C01828=1213.593,-33.093,-40.651,-179.967,5.450,148.943
C01829=1213.588,-32.844,-40.663,-179.964,5.451,148.942
C01830=1213.583,-32.594,-40.675,-179.962,5.450,148.942
C01831=1213.578,-32.344,-40.688,-179.960,5.451,148.941
C01832=1213.572,-32.095,-40.701,-179.957,5.451,148.940
C01833=1213.567,-31.845,-40.714,-179.955,5.451,148.940
C01834=1213.563,-31.595,-40.727,-179.953,5.452,148.939
C01835=1213.558,-31.347,-40.740,-179.950,5.452,148.939
C01836=1213.552,-31.097,-40.753,-179.948,5.452,148.938
C01837=1213.548,-30.847,-40.766,-179.945,5.452,148.937
C01838=1213.542,-30.598,-40.779,-179.943,5.453,148.936
C01839=1213.537,-30.348,-40.791,-179.941,5.453,148.936
C01840=1213.532,-30.098,-40.805,-179.938,5.453,148.935
C01841=1213.527,-29.849,-40.818,-179.935,5.454,148.934
C01842=1213.522,-29.599,-40.830,-179.933,5.454,148.934
C01843=1213.517,-29.349,-40.844,-179.931,5.454,148.933
C01844=1213.511,-29.100,-40.856,-179.928,5.454,148.932
C01845=1213.506,-28.850,-40.869,-179.925,5.455,148.932
C01846=1213.501,-28.600,-40.883,-179.923,5.454,148.931
C01847=1213.496,-28.351,-40.895,-179.921,5.455,148.930
C01848=1213.491,-28.101,-40.908,-179.918,5.456,148.930
C01849=1213.486,-27.852,-40.922,-179.916,5.455,148.929
C01850=1213.481,-27.602,-40.935,-179.914,5.456,148.928
C01851=1213.476,-27.352,-40.948,-179.911,5.456,148.928
C01852=1213.470,-27.103,-40.961,-179.908,5.457,148.927
C01853=1213.465,-26.853,-40.973,-179.906,5.456,148.926
C01854=1213.461,-26.603,-40.986,-179.904,5.457,148.925
C01855=1213.455,-26.354,-41.000,-179.901,5.457,148.925
C01856=1213.451,-26.104,-41.013,-179.899,5.457,148.924
C01857=1213.446,-25.855,-41.026,-179.896,5.458,148.923
C01858=1213.440,-25.605,-41.039,-179.893,5.458,148.923
C01859=1213.435,-25.355,-41.052,-179.891,5.458,148.922
C01860=1213.429,-25.106,-41.065,-179.889,5.458,148.921
C01861=1213.425,-24.856,-41.079,-179.887,5.459,148.921
C01862=1213.420,-24.607,-41.091,-179.884,5.460,148.920
C01863=1213.414,-24.357,-41.105,-179.882,5.459,148.919
C01864=1213.410,-24.107,-41.118,-179.879,5.460,148.919
C01865=1213.404,-23.858,-41.132,-179.877,5.460,148.918
C01866=1213.399,-23.608,-41.145,-179.874,5.460,148.917
C01867=1213.394,-23.359,-41.157,-179.872,5.460,148.917
C01868=1213.389,-23.090,-41.172,-179.869,5.461,148.916
C01869=1213.383,-22.820,-41.186,-179.866,5.461,148.915
C01870=1213.378,-22.551,-41.200,-179.863,5.462,148.914
C01871=1213.372,-22.281,-41.215,-179.861,5.462,148.914
C01872=1213.368,-22.031,-41.228,-179.859,5.462,148.913
C01873=1213.362,-21.782,-41.242,-179.856,5.462,148.912
C01874=1213.357,-21.533,-41.254,-179.854,5.463,148.912
C01875=1213.352,-21.282,-41.268,-179.852,5.463,148.911
C01876=1213.347,-21.034,-41.281,-179.849,5.463,148.910
C01877=1213.342,-20.783,-41.295,-179.846,5.464,148.910
C01878=1213.336,-20.534,-41.307,-179.844,5.464,148.909
C01879=1213.332,-20.284,-41.321,-179.842,5.464,148.908
C01880=1213.326,-20.035,-41.334,-179.839,5.464,148.908
C01881=1213.321,-19.785,-41.348,-179.836,5.465,148.907
C01882=1213.316,-19.536,-41.361,-179.834,5.465,148.906
C01883=1213.311,-19.286,-41.375,-179.832,5.465,148.906
C01884=1213.306,-19.037,-41.388,-179.829,5.466,148.905
C01885=1213.301,-18.787,-41.401,-179.826,5.466,148.904
C01886=1213.295,-18.537,-41.415,-179.824,5.466,148.903
C01887=1213.291,-18.288,-41.428,-179.822,5.466,148.903
C01888=1213.285,-18.038,-41.441,-179.819,5.467,148.902
C01889=1213.281,-17.789,-41.455,-179.817,5.468,148.902
C01890=1213.275,-17.539,-41.468,-179.815,5.467,148.901
C01891=1213.270,-17.289,-41.481,-179.812,5.468,148.900
C01892=1213.265,-17.040,-41.495,-179.809,5.468,148.900
C01893=1213.260,-16.790,-41.508,-179.807,5.469,148.899
C01894=1213.255,-16.541,-41.522,-179.805,5.468,148.898
C01895=1213.250,-16.291,-41.536,-179.802,5.469,148.897
C01896=1213.245,-16.041,-41.549,-179.799,5.469,148.897
C01897=1213.239,-15.792,-41.563,-179.797,5.470,148.896
C01898=1213.235,-15.542,-41.576,-179.794,5.470,148.895
C01899=1213.229,-15.293,-41.589,-179.792,5.470,148.895
C01900=1213.224,-15.043,-41.604,-179.789,5.471,148.894
C01901=1213.219,-14.794,-41.616,-179.787,5.471,148.893
C01902=1213.214,-14.544,-41.631,-179.785,5.471,148.893
C01903=1213.208,-14.294,-41.644,-179.782,5.472,148.892
C01904=1213.204,-14.045,-41.657,-179.780,5.472,148.891
C01905=1213.199,-13.795,-41.672,-179.777,5.473,148.891
C01906=1213.194,-13.546,-41.684,-179.775,5.472,148.890
C01907=1213.189,-13.296,-41.699,-179.772,5.473,148.889
C01908=1213.183,-13.046,-41.712,-179.770,5.473,148.889
C01909=1213.179,-12.797,-41.725,-179.767,5.474,148.888
C01910=1213.174,-12.547,-41.739,-179.765,5.473,148.887
C01911=1213.168,-12.298,-41.753,-179.762,5.474,148.887
C01912=1213.164,-12.048,-41.767,-179.760,5.474,148.886
C01913=1213.158,-11.799,-41.780,-179.757,5.475,148.885
C01914=1213.153,-11.549,-41.794,-179.755,5.475,148.885
C01915=1213.149,-11.300,-41.808,-179.753,5.475,148.884
C01916=1213.143,-11.050,-41.821,-179.750,5.476,148.883
C01917=1213.138,-10.800,-41.835,-179.747,5.476,148.883
C01918=1213.132,-10.551,-41.848,-179.745,5.477,148.882
C01919=1213.128,-10.301,-41.862,-179.743,5.477,148.881
C01920=1213.123,-10.051,-41.876,-179.740,5.477,148.881
C01921=1213.117,-9.802,-41.890,-179.737,5.478,148.880
C01922=1213.113,-9.552,-41.903,-179.735,5.478,148.879
C01923=1213.108,-9.303,-41.918,-179.733,5.478,148.878
C01924=1213.103,-9.054,-41.931,-179.730,5.478,148.878
C01925=1213.097,-8.803,-41.945,-179.727,5.479,148.877
C01926=1213.093,-8.554,-41.959,-179.725,5.479,148.876
C01927=1213.088,-8.305,-41.973,-179.723,5.479,148.876
C01928=1213.082,-8.055,-41.986,-179.720,5.480,148.875
C01929=1213.077,-7.805,-42.000,-179.718,5.480,148.875
C01930=1213.072,-7.556,-42.014,-179.715,5.481,148.874
C01931=1213.068,-7.307,-42.028,-179.712,5.481,148.873
C01932=1213.062,-7.056,-42.042,-179.710,5.481,148.872
C01933=1213.057,-6.807,-42.056,-179.708,5.482,148.872
C01934=1213.052,-6.557,-42.070,-179.705,5.482,148.871
C01935=1213.048,-6.308,-42.084,-179.702,5.483,148.870
C01936=1213.042,-6.059,-42.097,-179.700,5.482,148.870
C01937=1213.037,-5.809,-42.111,-179.698,5.483,148.869
C01938=1213.032,-5.559,-42.125,-179.695,5.483,148.868
C01939=1213.027,-5.309,-42.140,-179.693,5.484,148.868
C01940=1213.021,-5.060,-42.153,-179.690,5.485,148.867
C01941=1213.017,-4.811,-42.167,-179.688,5.484,148.867
C01942=1213.012,-4.561,-42.181,-179.685,5.485,148.866
C01943=1213.006,-4.312,-42.195,-179.683,5.485,148.865
C01944=1213.001,-4.062,-42.209,-179.680,5.486,148.864
C01945=1212.996,-3.812,-42.223,-179.677,5.486,148.864
C01946=1212.991,-3.562,-42.237,-179.675,5.486,148.863
C01947=1212.986,-3.313,-42.251,-179.673,5.487,148.862
C01948=1212.982,-3.064,-42.265,-179.670,5.487,148.862
C01949=1212.977,-2.814,-42.279,-179.667,5.488,148.861
C01950=1212.971,-2.565,-42.293,-179.665,5.488,148.861
C01951=1212.966,-2.315,-42.307,-179.663,5.488,148.860
C01952=1212.961,-2.065,-42.321,-179.660,5.489,148.859
C01953=1212.956,-1.816,-42.335,-179.658,5.489,148.858
C01954=1212.950,-1.567,-42.349,-179.655,5.490,148.858
C01955=1212.945,-1.317,-42.364,-179.653,5.490,148.857
C01956=1212.941,-1.067,-42.378,-179.650,5.490,148.856
C01957=1212.936,-0.817,-42.392,-179.648,5.490,148.856
C01958=1212.931,-0.568,-42.406,-179.645,5.491,148.855
C01959=1212.926,-0.319,-42.420,-179.642,5.491,148.854
C01960=1212.921,-0.069,-42.434,-179.640,5.492,148.854
C01961=1212.916,0.180,-42.448,-179.638,5.492,148.853
C01962=1212.911,0.430,-42.462,-179.636,5.492,148.852
C01963=1212.905,0.679,-42.476,-179.633,5.493,148.852
C01964=1212.900,0.929,-42.491,-179.630,5.493,148.851
C01965=1212.895,1.179,-42.505,-179.628,5.494,148.850
C01966=1212.891,1.428,-42.519,-179.626,5.494,148.850
C01967=1212.886,1.678,-42.534,-179.623,5.494,148.849
C01968=1212.880,1.927,-42.547,-179.620,5.495,148.848
C01969=1212.875,2.177,-42.562,-179.618,5.495,148.848
C01970=1212.870,2.426,-42.576,-179.615,5.496,148.847
C01971=1212.865,2.676,-42.590,-179.612,5.496,148.846
C01972=1212.860,2.945,-42.606,-179.610,5.496,148.846
C01973=1212.855,3.214,-42.621,-179.608,5.496,148.845
C01974=1212.848,3.483,-42.637,-179.605,5.497,148.844
C01975=1212.843,3.751,-42.653,-179.602,5.497,148.844
C01976=1212.838,4.001,-42.667,-179.600,5.498,148.843
C01977=1212.833,4.251,-42.681,-179.597,5.498,148.842
C01978=1212.828,4.501,-42.695,-179.594,5.499,148.841
C01979=1212.823,4.750,-42.710,-179.592,5.499,148.841
C01980=1212.818,5.000,-42.724,-179.590,5.499,148.840
C01981=1212.813,5.249,-42.738,-179.587,5.500,148.840
C01982=1212.808,5.499,-42.752,-179.585,5.501,148.839
C01983=1212.803,5.748,-42.767,-179.582,5.501,148.838
C01984=1212.798,5.998,-42.781,-179.579,5.502,148.838
C01985=1212.793,6.247,-42.796,-179.577,5.502,148.837
C01986=1212.788,6.497,-42.810,-179.575,5.502,148.836
C01987=1212.783,6.747,-42.824,-179.572,5.502,148.836
C01988=1212.777,6.995,-42.840,-179.569,5.503,148.835
C01989=1212.772,7.245,-42.854,-179.567,5.503,148.834
C01990=1212.767,7.495,-42.868,-179.564,5.504,148.833
C01991=1212.762,7.745,-42.882,-179.562,5.505,148.833
C01992=1212.758,7.994,-42.897,-179.559,5.505,148.832
C01993=1212.753,8.243,-42.912,-179.557,5.505,148.832
C01994=1212.748,8.493,-42.926,-179.555,5.505,148.831
C01995=1212.743,8.743,-42.940,-179.552,5.506,148.830
C01996=1212.737,8.992,-42.956,-179.549,5.507,148.830
C01997=1212.733,9.242,-42.970,-179.547,5.507,148.829
C01998=1212.728,9.492,-42.984,-179.544,5.508,148.828
C01999=1212.722,9.741,-42.998,-179.542,5.507,148.828
C02000=1212.717,9.990,-43.013,-179.540,5.508,148.827
C02001=1212.712,10.239,-43.027,-179.537,5.509,148.826
C02002=1212.707,10.489,-43.042,-179.534,5.509,148.826
C02003=1212.702,10.739,-43.057,-179.532,5.510,148.825
C02004=1212.697,10.988,-43.072,-179.529,5.510,148.824
C02005=1212.692,11.238,-43.086,-179.527,5.511,148.824
C02006=1212.688,11.487,-43.101,-179.524,5.510,148.823
C02007=1212.682,11.737,-43.116,-179.522,5.511,148.822
C02008=1212.677,11.987,-43.130,-179.519,5.511,148.822
C02009=1212.672,12.236,-43.145,-179.517,5.512,148.821
C02010=1212.667,12.486,-43.159,-179.514,5.513,148.820
C02011=1212.663,12.735,-43.174,-179.512,5.513,148.820
C02012=1212.657,12.985,-43.189,-179.509,5.514,148.819
C02013=1212.652,13.234,-43.203,-179.507,5.514,148.818
C02014=1212.647,13.483,-43.218,-179.504,5.514,148.818
C02015=1212.642,13.733,-43.233,-179.502,5.515,148.817
C02016=1212.637,13.983,-43.248,-179.499,5.515,148.816
C02017=1212.632,14.232,-43.263,-179.496,5.516,148.816
C02018=1212.627,14.481,-43.278,-179.494,5.517,148.815
C02019=1212.622,14.731,-43.292,-179.492,5.517,148.815
C02020=1212.617,14.981,-43.307,-179.490,5.517,148.814
C02021=1212.612,15.230,-43.322,-179.487,5.517,148.813
C02022=1212.607,15.480,-43.336,-179.484,5.518,148.812
C02023=1212.602,15.729,-43.352,-179.482,5.518,148.812
C02024=1212.597,15.979,-43.366,-179.479,5.519,148.811
C02025=1212.592,16.228,-43.381,-179.476,5.519,148.810
C02026=1212.586,16.478,-43.396,-179.474,5.520,148.810
C02027=1212.582,16.727,-43.411,-179.471,5.521,148.809
C02028=1212.577,16.977,-43.425,-179.469,5.520,148.809
C02029=1212.571,17.226,-43.441,-179.467,5.521,148.808
C02030=1212.567,17.475,-43.456,-179.464,5.522,148.807
C02031=1212.562,17.725,-43.470,-179.461,5.522,148.807
C02032=1212.556,17.975,-43.485,-179.459,5.523,148.806
C02033=1212.552,18.224,-43.500,-179.456,5.523,148.805
C02034=1212.547,18.473,-43.515,-179.454,5.524,148.805
C02035=1212.541,18.723,-43.530,-179.451,5.525,148.804
C02036=1212.537,18.972,-43.545,-179.449,5.525,148.803
C02037=1212.532,19.222,-43.560,-179.447,5.525,148.803
C02038=1212.526,19.472,-43.574,-179.444,5.525,148.802
C02039=1212.522,19.721,-43.589,-179.441,5.526,148.801
C02040=1212.516,19.971,-43.604,-179.439,5.526,148.801
C02041=1212.512,20.220,-43.620,-179.436,5.527,148.800
C02042=1212.507,20.470,-43.635,-179.434,5.528,148.800
C02043=1212.501,20.720,-43.650,-179.431,5.528,148.799
C02044=1212.497,20.969,-43.665,-179.429,5.529,148.798
C02045=1212.491,21.218,-43.680,-179.426,5.529,148.797
C02046=1212.486,21.468,-43.694,-179.423,5.530,148.797
C02047=1212.481,21.717,-43.710,-179.421,5.530,148.796
C02048=1212.476,21.966,-43.725,-179.419,5.530,148.795
C02049=1212.471,22.216,-43.739,-179.416,5.531,148.795
C02050=1212.466,22.465,-43.755,-179.414,5.531,148.794
C02051=1212.462,22.715,-43.770,-179.411,5.532,148.794
C02052=1212.457,22.965,-43.786,-179.408,5.533,148.793
C02053=1212.452,23.214,-43.800,-179.406,5.533,148.792
C02054=1212.446,23.464,-43.816,-179.403,5.534,148.792
C02055=1212.442,23.713,-43.831,-179.401,5.534,148.791
C02056=1212.436,23.962,-43.846,-179.398,5.535,148.790
C02057=1212.431,24.212,-43.861,-179.396,5.535,148.790
C02058=1212.426,24.461,-43.876,-179.394,5.535,148.789
C02059=1212.422,24.711,-43.891,-179.391,5.536,148.788
C02060=1212.416,24.961,-43.907,-179.388,5.536,148.788
C02061=1212.412,25.210,-43.921,-179.386,5.537,148.787
C02062=1212.406,25.460,-43.937,-179.383,5.537,148.786
C02063=1212.401,25.709,-43.952,-179.380,5.538,148.786
C02064=1212.396,25.958,-43.967,-179.378,5.539,148.785
C02065=1212.392,26.208,-43.983,-179.376,5.539,148.785
C02066=1212.387,26.457,-43.998,-179.373,5.540,148.784
C02067=1212.381,26.707,-44.013,-179.370,5.540,148.783
C02068=1212.376,26.956,-44.028,-179.368,5.541,148.783
C02069=1212.371,27.206,-44.044,-179.365,5.541,148.782
C02070=1212.367,27.456,-44.059,-179.363,5.541,148.781
C02071=1212.362,27.705,-44.075,-179.361,5.542,148.781
C02072=1212.357,27.954,-44.090,-179.358,5.543,148.780
C02073=1212.351,28.204,-44.105,-179.356,5.543,148.779
C02074=1212.346,28.453,-44.121,-179.353,5.544,148.779
C02075=1212.342,28.703,-44.136,-179.350,5.544,148.778
C02076=1212.336,28.972,-44.153,-179.348,5.545,148.777
C02077=1212.331,29.240,-44.170,-179.345,5.545,148.777
C02078=1212.325,29.509,-44.185,-179.342,5.546,148.776
C02079=1212.320,29.778,-44.202,-179.340,5.546,148.775
C02080=1212.315,30.027,-44.218,-179.337,5.547,148.775
C02081=1212.310,30.276,-44.233,-179.334,5.547,148.774
C02082=1212.305,30.526,-44.249,-179.332,5.548,148.773
C02083=1212.300,30.775,-44.264,-179.329,5.548,148.773
C02084=1212.295,31.025,-44.280,-179.327,5.549,148.772
C02085=1212.290,31.274,-44.295,-179.324,5.550,148.771
C02086=1212.286,31.524,-44.310,-179.322,5.550,148.771
C02087=1212.280,31.773,-44.326,-179.319,5.551,148.770
C02088=1212.275,32.023,-44.342,-179.316,5.551,148.769
C02089=1212.270,32.272,-44.357,-179.314,5.552,148.769
C02090=1212.265,32.522,-44.373,-179.312,5.553,148.768
C02091=1212.260,32.771,-44.388,-179.309,5.553,148.768
C02092=1212.255,33.021,-44.404,-179.306,5.554,148.767
C02093=1212.250,33.270,-44.419,-179.304,5.554,148.766
C02094=1212.245,33.520,-44.435,-179.301,5.555,148.766
C02095=1212.240,33.769,-44.450,-179.298,5.556,148.765
C02096=1212.235,34.018,-44.465,-179.296,5.556,148.764
C02097=1212.230,34.268,-44.481,-179.294,5.557,148.764
C02098=1212.225,34.517,-44.498,-179.291,5.557,148.763
C02099=1212.220,34.767,-44.513,-179.289,5.557,148.762
C02100=1212.215,35.016,-44.528,-179.286,5.558,148.762
C02101=1212.210,35.266,-44.544,-179.284,5.558,148.761
C02102=1212.205,35.515,-44.560,-179.281,5.559,148.761
C02103=1212.200,35.765,-44.575,-179.279,5.560,148.760
C02104=1212.196,36.014,-44.591,-179.276,5.560,148.759
C02105=1212.191,36.263,-44.607,-179.273,5.561,148.759
C02106=1212.185,36.513,-44.623,-179.271,5.561,148.758
C02107=1212.180,36.763,-44.638,-179.268,5.562,148.757
C02108=1212.175,37.012,-44.654,-179.266,5.563,148.757
C02109=1212.170,37.261,-44.669,-179.263,5.563,148.756
C02110=1212.166,37.511,-44.685,-179.261,5.564,148.755
C02111=1212.161,37.760,-44.701,-179.258,5.564,148.755
C02112=1212.155,38.009,-44.717,-179.255,5.565,148.754
C02113=1212.150,38.260,-44.733,-179.253,5.565,148.753
C02114=1212.146,38.509,-44.748,-179.251,5.566,148.753
C02115=1212.141,38.757,-44.764,-179.248,5.567,148.752
C02116=1212.136,39.008,-44.780,-179.245,5.567,148.752
C02117=1212.130,39.257,-44.796,-179.243,5.568,148.751
C02118=1212.126,39.507,-44.812,-179.240,5.569,148.750
C02119=1212.121,39.756,-44.828,-179.238,5.569,148.750
C02120=1212.115,40.005,-44.844,-179.235,5.570,148.749
C02121=1212.111,40.255,-44.859,-179.233,5.571,148.749
C02122=1212.106,40.504,-44.875,-179.230,5.571,148.748
C02123=1212.101,40.753,-44.891,-179.227,5.572,148.747
C02124=1212.096,41.003,-44.907,-179.225,5.572,148.746
C02125=1212.091,41.252,-44.923,-179.223,5.573,148.746
C02126=1212.086,41.502,-44.939,-179.220,5.574,148.745
C02127=1212.081,41.752,-44.955,-179.217,5.574,148.745
C02128=1212.076,42.000,-44.971,-179.215,5.575,148.744
C02129=1212.071,42.251,-44.987,-179.212,5.575,148.743
C02130=1212.065,42.500,-45.002,-179.210,5.576,148.743
C02131=1212.062,42.749,-45.018,-179.207,5.577,148.742
C02132=1212.056,42.999,-45.034,-179.205,5.577,148.742
C02133=1212.052,43.248,-45.051,-179.202,5.578,148.741
C02134=1212.046,43.497,-45.066,-179.199,5.578,148.740
C02135=1212.041,43.747,-45.082,-179.197,5.579,148.740
C02136=1212.037,43.996,-45.099,-179.195,5.580,148.739
C02137=1212.031,44.246,-45.114,-179.192,5.580,148.738
C02138=1212.027,44.495,-45.131,-179.189,5.581,148.738
C02139=1212.021,44.745,-45.146,-179.187,5.581,148.737
C02140=1212.017,44.994,-45.163,-179.184,5.582,148.736
C02141=1212.011,45.243,-45.179,-179.182,5.583,148.736
C02142=1212.007,45.494,-45.195,-179.179,5.583,148.735
C02143=1212.002,45.742,-45.211,-179.177,5.584,148.735
C02144=1211.997,45.992,-45.227,-179.174,5.584,148.734
C02145=1211.992,46.241,-45.243,-179.171,5.585,148.733
C02146=1211.987,46.491,-45.259,-179.169,5.586,148.733
C02147=1211.982,46.740,-45.275,-179.167,5.586,148.732
C02148=1211.977,46.989,-45.292,-179.164,5.587,148.732
C02149=1211.972,47.239,-45.308,-179.161,5.588,148.731
C02150=1211.967,47.488,-45.324,-179.159,5.588,148.730
C02151=1211.962,47.738,-45.340,-179.156,5.589,148.730
C02152=1211.957,47.987,-45.356,-179.154,5.590,148.729
C02153=1211.952,48.237,-45.372,-179.151,5.590,148.728
C02154=1211.948,48.486,-45.389,-179.149,5.591,148.728
C02155=1211.942,48.736,-45.405,-179.146,5.592,148.727
C02156=1211.937,48.985,-45.422,-179.144,5.592,148.727
C02157=1211.932,49.234,-45.438,-179.141,5.593,148.726
C02158=1211.927,49.484,-45.454,-179.138,5.593,148.725
C02159=1211.922,49.733,-45.470,-179.136,5.594,148.725
C02160=1211.918,49.983,-45.487,-179.134,5.595,148.724
C02161=1211.912,50.232,-45.503,-179.131,5.595,148.723
C02162=1211.908,50.481,-45.519,-179.128,5.596,148.723
C02163=1211.902,50.731,-45.535,-179.126,5.596,148.722
C02164=1211.898,50.980,-45.552,-179.123,5.597,148.721
C02165=1211.892,51.229,-45.568,-179.120,5.599,148.721
C02166=1211.887,51.480,-45.584,-179.118,5.599,148.720
C02167=1211.883,51.729,-45.601,-179.115,5.600,148.720
C02168=1211.878,51.978,-45.617,-179.113,5.600,148.719
C02169=1211.873,52.227,-45.634,-179.110,5.601,148.719
C02170=1211.868,52.477,-45.650,-179.108,5.602,148.718
C02171=1211.863,52.726,-45.666,-179.105,5.602,148.717
C02172=1211.858,52.975,-45.683,-179.102,5.603,148.717
C02173=1211.853,53.225,-45.700,-179.100,5.603,148.716
C02174=1211.848,53.475,-45.716,-179.098,5.604,148.715
C02175=1211.843,53.724,-45.732,-179.095,5.605,148.715
C02176=1211.839,53.973,-45.749,-179.092,5.605,148.714
C02177=1211.833,54.222,-45.766,-179.090,5.606,148.713
C02178=1211.828,54.472,-45.782,-179.088,5.607,148.713
C02179=1211.824,54.722,-45.798,-179.085,5.607,148.712
C02180=1211.818,54.990,-45.816,-179.082,5.608,148.712
C02181=1211.812,55.258,-45.834,-179.079,5.609,148.711
C02182=1211.808,55.527,-45.852,-179.077,5.610,148.710
C02183=1211.802,55.795,-45.869,-179.074,5.610,148.710
C02184=1211.798,56.044,-45.886,-179.071,5.611,148.709
C02185=1211.792,56.295,-45.903,-179.069,5.612,148.708
C02186=1211.787,56.544,-45.919,-179.066,5.612,148.708
C02187=1211.783,56.793,-45.936,-179.064,5.613,148.707
C02188=1211.778,57.042,-45.952,-179.061,5.614,148.707
C02189=1211.772,57.292,-45.969,-179.058,5.615,148.706
C02190=1211.768,57.541,-45.986,-179.055,5.615,148.705
C02191=1211.763,57.790,-46.002,-179.053,5.616,148.705
C02192=1211.758,58.040,-46.019,-179.051,5.617,148.704
C02193=1211.753,58.290,-46.035,-179.048,5.617,148.704
C02194=1211.748,58.539,-46.052,-179.045,5.618,148.703
C02195=1211.743,58.788,-46.069,-179.043,5.619,148.702
C02196=1211.738,59.038,-46.086,-179.041,5.620,148.702
C02197=1211.733,59.287,-46.102,-179.038,5.620,148.701
C02198=1211.728,59.536,-46.119,-179.035,5.621,148.700
C02199=1211.723,59.786,-46.136,-179.033,5.622,148.700
C02200=1211.719,60.035,-46.153,-179.030,5.622,148.699
C02201=1211.713,60.285,-46.169,-179.028,5.623,148.699
C02202=1211.708,60.534,-46.186,-179.025,5.624,148.698
C02203=1211.704,60.784,-46.203,-179.023,5.625,148.698
C02204=1211.698,61.033,-46.220,-179.020,5.626,148.697
C02205=1211.694,61.282,-46.236,-179.017,5.626,148.696
C02206=1211.689,61.532,-46.253,-179.015,5.627,148.696
C02207=1211.683,61.781,-46.270,-179.012,5.628,148.695
C02208=1211.679,62.030,-46.287,-179.010,5.628,148.694
C02209=1211.674,62.280,-46.304,-179.007,5.629,148.694
C02210=1211.669,62.529,-46.321,-179.005,5.629,148.693
C02211=1211.664,62.778,-46.337,-179.002,5.630,148.693
C02212=1211.659,63.028,-46.354,-178.999,5.632,148.692
C02213=1211.655,63.277,-46.371,-178.997,5.632,148.691
C02214=1211.650,63.527,-46.389,-178.994,5.633,148.691
C02215=1211.644,63.775,-46.405,-178.992,5.634,148.690
C02216=1211.639,64.025,-46.422,-178.989,5.634,148.690
C02217=1211.635,64.275,-46.439,-178.987,5.635,148.689
C02218=1211.630,64.524,-46.456,-178.984,5.636,148.689
C02219=1211.624,64.773,-46.473,-178.982,5.636,148.688
C02220=1211.620,65.023,-46.489,-178.979,5.637,148.687
C02221=1211.615,65.272,-46.507,-178.977,5.637,148.687
C02222=1211.611,65.521,-46.524,-178.974,5.639,148.686
C02223=1211.605,65.771,-46.541,-178.971,5.640,148.685
C02224=1211.600,66.020,-46.557,-178.969,5.640,148.685
C02225=1211.595,66.270,-46.575,-178.966,5.641,148.684
C02226=1211.591,66.519,-46.592,-178.964,5.642,148.684
C02227=1211.586,66.768,-46.609,-178.961,5.642,148.683
C02228=1211.581,67.018,-46.626,-178.959,5.643,148.682
C02229=1211.575,67.267,-46.643,-178.956,5.644,148.682
C02230=1211.571,67.517,-46.660,-178.953,5.645,148.681
C02231=1211.566,67.766,-46.678,-178.951,5.646,148.681
C02232=1211.562,68.015,-46.694,-178.948,5.646,148.680
C02233=1211.556,68.265,-46.711,-178.946,5.647,148.679
C02234=1211.552,68.513,-46.729,-178.943,5.648,148.679
C02235=1211.546,68.763,-46.746,-178.941,5.648,148.678
C02236=1211.541,69.013,-46.763,-178.938,5.649,148.678
C02237=1211.537,69.262,-46.780,-178.936,5.650,148.677
C02238=1211.532,69.511,-46.798,-178.933,5.651,148.676
C02239=1211.527,69.761,-46.814,-178.930,5.652,148.676
C02240=1211.522,70.011,-46.832,-178.928,5.653,148.675
C02241=1211.517,70.259,-46.849,-178.925,5.653,148.675
C02242=1211.512,70.509,-46.866,-178.923,5.654,148.674
C02243=1211.507,70.758,-46.883,-178.920,5.654,148.673
C02244=1211.503,71.007,-46.901,-178.918,5.655,148.673
C02245=1211.497,71.257,-46.918,-178.915,5.657,148.672
C02246=1211.492,71.507,-46.935,-178.912,5.657,148.672
C02247=1211.488,71.756,-46.952,-178.910,5.658,148.671
C02248=1211.482,72.005,-46.969,-178.907,5.659,148.671
C02249=1211.478,72.254,-46.987,-178.905,5.659,148.670
C02250=1211.473,72.504,-47.004,-178.902,5.660,148.669
C02251=1211.468,72.753,-47.022,-178.900,5.661,148.669
C02252=1211.463,73.002,-47.039,-178.897,5.662,148.668
C02253=1211.458,73.252,-47.056,-178.894,5.663,148.667
C02254=1211.453,73.501,-47.074,-178.892,5.664,148.667
C02255=1211.449,73.751,-47.091,-178.889,5.664,148.666
C02256=1211.444,74.000,-47.109,-178.887,5.665,148.666
C02257=1211.439,74.250,-47.126,-178.884,5.666,148.665
C02258=1211.434,74.499,-47.144,-178.881,5.667,148.665
C02259=1211.429,74.748,-47.160,-178.879,5.668,148.664
C02260=1211.424,74.997,-47.178,-178.876,5.669,148.664
C02261=1211.419,75.247,-47.195,-178.874,5.669,148.663
C02262=1211.414,75.495,-47.213,-178.871,5.670,148.662
C02263=1211.409,75.745,-47.230,-178.869,5.670,148.662
C02264=1211.404,75.994,-47.248,-178.866,5.672,148.661
C02265=1211.399,76.244,-47.265,-178.863,5.673,148.660
C02266=1211.395,76.493,-47.283,-178.861,5.673,148.660
C02267=1211.390,76.742,-47.301,-178.858,5.674,148.659
C02268=1211.385,76.992,-47.318,-178.856,5.675,148.659
C02269=1211.380,77.241,-47.336,-178.853,5.675,148.658
C02270=1211.375,77.491,-47.353,-178.850,5.677,148.658
C02271=1211.370,77.740,-47.370,-178.848,5.677,148.657
C02272=1211.366,77.989,-47.388,-178.845,5.678,148.656
C02273=1211.360,78.239,-47.406,-178.843,5.679,148.656
C02274=1211.355,78.488,-47.424,-178.840,5.680,148.655
C02275=1211.351,78.737,-47.440,-178.837,5.681,148.655
C02276=1211.346,78.987,-47.458,-178.835,5.682,148.654
C02277=1211.341,79.236,-47.476,-178.832,5.682,148.654
C02278=1211.336,79.486,-47.494,-178.830,5.683,148.653
C02279=1211.331,79.735,-47.512,-178.828,5.684,148.652
C02280=1211.327,79.984,-47.529,-178.825,5.685,148.652
C02281=1211.322,80.233,-47.546,-178.822,5.686,148.651
C02282=1211.317,80.483,-47.564,-178.820,5.687,148.651
C02283=1211.312,80.732,-47.582,-178.817,5.687,148.650
C02284=1211.306,81.001,-47.601,-178.815,5.688,148.649
C02285=1211.301,81.269,-47.620,-178.811,5.689,148.649
C02286=1211.296,81.536,-47.639,-178.809,5.690,148.648
C02287=1211.290,81.805,-47.658,-178.805,5.691,148.647
C02288=1211.285,82.055,-47.676,-178.803,5.692,148.647
C02289=1211.280,82.304,-47.694,-178.801,5.693,148.646
C02290=1211.276,82.554,-47.712,-178.798,5.693,148.646
C02291=1211.272,82.803,-47.729,-178.796,5.694,148.645
C02292=1211.267,83.052,-47.747,-178.793,5.696,148.645
C02293=1211.262,83.301,-47.765,-178.790,5.696,148.644
C02294=1211.257,83.551,-47.783,-178.788,5.697,148.644
C02295=1211.252,83.800,-47.801,-178.785,5.698,148.643
C02296=1211.247,84.050,-47.818,-178.783,5.699,148.642
C02297=1211.242,84.299,-47.836,-178.780,5.700,148.642
C02298=1211.237,84.548,-47.854,-178.777,5.701,148.641
C02299=1211.232,84.797,-47.872,-178.775,5.702,148.641
C02300=1211.227,85.046,-47.890,-178.773,5.702,148.640
C02301=1211.222,85.295,-47.908,-178.769,5.704,148.639
C02302=1211.217,85.545,-47.926,-178.767,5.705,148.639
C02303=1211.213,85.794,-47.944,-178.765,5.705,148.638
C02304=1211.208,86.044,-47.962,-178.762,5.706,148.638
C02305=1211.203,86.293,-47.980,-178.760,5.707,148.637
C02306=1211.198,86.543,-47.998,-178.757,5.708,148.637
C02307=1211.193,86.792,-48.016,-178.754,5.709,148.636
C02308=1211.188,87.041,-48.034,-178.752,5.710,148.636
C02309=1211.183,87.290,-48.052,-178.749,5.710,148.635
C02310=1211.178,87.539,-48.070,-178.747,5.712,148.635
C02311=1211.174,87.789,-48.088,-178.744,5.713,148.634
C02312=1211.169,88.038,-48.106,-178.741,5.713,148.633
C02313=1211.164,88.288,-48.124,-178.739,5.714,148.633
C02314=1211.159,88.537,-48.142,-178.736,5.715,148.632
C02315=1211.154,88.786,-48.160,-178.734,5.716,148.631
C02316=1211.149,89.035,-48.178,-178.731,5.717,148.631
C02317=1211.144,89.284,-48.196,-178.729,5.718,148.630
C02318=1211.140,89.534,-48.214,-178.726,5.719,148.630
C02319=1211.135,89.783,-48.232,-178.723,5.720,148.629
C02320=1211.130,90.032,-48.250,-178.721,5.720,148.629
C02321=1211.125,90.282,-48.269,-178.719,5.721,148.628
C02322=1211.120,90.531,-48.287,-178.715,5.723,148.628
C02323=1211.115,90.780,-48.305,-178.713,5.723,148.627
C02324=1211.111,91.030,-48.323,-178.711,5.724,148.627
C02325=1211.106,91.279,-48.342,-178.708,5.725,148.626
C02326=1211.101,91.528,-48.360,-178.705,5.726,148.625
C02327=1211.096,91.777,-48.378,-178.703,5.727,148.625
C02328=1211.091,92.026,-48.396,-178.700,5.728,148.624
C02329=1211.086,92.276,-48.415,-178.698,5.729,148.624
C02330=1211.081,92.526,-48.433,-178.695,5.730,148.623
C02331=1211.076,92.775,-48.451,-178.692,5.731,148.622
C02332=1211.071,93.024,-48.468,-178.690,5.732,148.622
C02333=1211.067,93.273,-48.488,-178.687,5.732,148.621
C02334=1211.062,93.522,-48.506,-178.685,5.734,148.621
C02335=1211.058,93.772,-48.524,-178.682,5.735,148.620
C02336=1211.052,94.021,-48.542,-178.680,5.735,148.620
C02337=1211.048,94.271,-48.560,-178.677,5.736,148.619
C02338=1211.043,94.520,-48.579,-178.674,5.738,148.619
C02339=1211.038,94.769,-48.597,-178.672,5.738,148.618
C02340=1211.032,95.018,-48.616,-178.669,5.739,148.618
C02341=1211.028,95.268,-48.634,-178.666,5.740,148.617
C02342=1211.024,95.517,-48.653,-178.664,5.741,148.617
C02343=1211.019,95.766,-48.671,-178.662,5.742,148.616
C02344=1211.014,96.015,-48.689,-178.659,5.743,148.615
C02345=1211.009,96.265,-48.708,-178.656,5.744,148.615
C02346=1211.004,96.514,-48.726,-178.654,5.745,148.614
C02347=1210.999,96.763,-48.744,-178.651,5.746,148.614
C02348=1210.994,97.012,-48.762,-178.648,5.747,148.613
C02349=1210.989,97.262,-48.782,-178.646,5.748,148.613
C02350=1210.985,97.511,-48.800,-178.644,5.749,148.612
C02351=1210.980,97.760,-48.818,-178.641,5.749,148.611
C02352=1210.975,98.010,-48.838,-178.638,5.751,148.611
C02353=1210.970,98.259,-48.856,-178.636,5.752,148.610
C02354=1210.965,98.508,-48.874,-178.633,5.753,148.610
C02355=1210.961,98.757,-48.893,-178.630,5.754,148.609
C02356=1210.955,99.007,-48.911,-178.628,5.755,148.609
C02357=1210.951,99.256,-48.929,-178.626,5.756,148.608
C02358=1210.947,99.505,-48.948,-178.622,5.757,148.608
C02359=1210.941,99.755,-48.967,-178.620,5.758,148.607
C02360=1210.936,100.003,-48.985,-178.618,5.759,148.606
C02361=1210.932,100.253,-49.004,-178.615,5.759,148.606
C02362=1210.926,100.503,-49.022,-178.612,5.761,148.605
C02363=1210.922,100.751,-49.041,-178.610,5.761,148.605
C02364=1210.917,101.001,-49.060,-178.608,5.762,148.604
C02365=1210.912,101.250,-49.079,-178.604,5.764,148.604
C02366=1210.907,101.499,-49.097,-178.602,5.765,148.603
C02367=1210.902,101.749,-49.116,-178.600,5.765,148.603
C02368=1210.897,101.998,-49.134,-178.597,5.767,148.602
C02369=1210.893,102.246,-49.153,-178.594,5.768,148.602
C02370=1210.888,102.496,-49.172,-178.592,5.768,148.601
C02371=1210.883,102.745,-49.191,-178.589,5.770,148.601
C02372=1210.878,102.995,-49.210,-178.586,5.771,148.600
C02373=1210.874,103.244,-49.228,-178.584,5.772,148.600
C02374=1210.868,103.493,-49.247,-178.581,5.773,148.599
C02375=1210.864,103.743,-49.266,-178.579,5.774,148.598
C02376=1210.859,103.991,-49.285,-178.576,5.775,148.598
C02377=1210.854,104.241,-49.304,-178.573,5.776,148.597
C02378=1210.850,104.490,-49.322,-178.571,5.777,148.597
C02379=1210.844,104.739,-49.341,-178.568,5.778,148.596
C02380=1210.840,104.989,-49.360,-178.566,5.779,148.596
C02381=1210.834,105.238,-49.378,-178.563,5.780,148.595
C02382=1210.830,105.487,-49.398,-178.561,5.781,148.595
C02383=1210.825,105.736,-49.417,-178.558,5.782,148.594
C02384=1210.821,105.986,-49.435,-178.556,5.783,148.594
C02385=1210.815,106.235,-49.454,-178.553,5.784,148.593
C02386=1210.811,106.483,-49.473,-178.550,5.786,148.593
C02387=1210.806,106.734,-49.492,-178.548,5.786,148.592
C02388=1210.800,107.002,-49.513,-178.545,5.787,148.591
C02389=1210.796,107.271,-49.533,-178.542,5.789,148.591
C02390=1210.790,107.538,-49.553,-178.540,5.789,148.590
C02391=1210.785,107.807,-49.574,-178.537,5.791,148.590
C02392=1210.780,108.056,-49.592,-178.534,5.791,148.589
C02393=1210.776,108.306,-49.612,-178.531,5.793,148.589
C02394=1210.771,108.554,-49.631,-178.529,5.793,148.588
C02395=1210.766,108.804,-49.650,-178.527,5.794,148.587
C02396=1210.761,109.054,-49.669,-178.523,5.796,148.587
C02397=1210.756,109.302,-49.688,-178.521,5.797,148.586
C02398=1210.751,109.552,-49.707,-178.518,5.798,148.586
C02399=1210.747,109.800,-49.726,-178.516,5.799,148.585
C02400=1210.742,110.050,-49.745,-178.513,5.800,148.585
C02401=1210.736,110.299,-49.764,-178.511,5.802,148.584
C02402=1210.732,110.548,-49.783,-178.508,5.802,148.584
C02403=1210.727,110.798,-49.803,-178.506,5.803,148.583
C02404=1210.723,111.047,-49.822,-178.503,5.804,148.583
C02405=1210.718,111.296,-49.841,-178.501,5.805,148.582
C02406=1210.712,111.546,-49.860,-178.498,5.806,148.582
C02407=1210.708,111.795,-49.879,-178.495,5.808,148.581
C02408=1210.703,112.044,-49.898,-178.493,5.808,148.581
C02409=1210.698,112.293,-49.918,-178.490,5.810,148.580
C02410=1210.694,112.542,-49.937,-178.487,5.811,148.580
C02411=1210.689,112.791,-49.956,-178.485,5.812,148.579
C02412=1210.684,113.040,-49.976,-178.482,5.813,148.579
C02413=1210.680,113.290,-49.995,-178.480,5.814,148.578
C02414=1210.674,113.538,-50.014,-178.477,5.815,148.577
C02415=1210.669,113.789,-50.033,-178.475,5.816,148.577
C02416=1210.665,114.038,-50.052,-178.472,5.817,148.576
C02417=1210.660,114.287,-50.071,-178.469,5.818,148.576
C02418=1210.655,114.536,-50.091,-178.467,5.819,148.575
C02419=1210.650,114.785,-50.110,-178.464,5.820,148.575
C02420=1210.646,115.034,-50.129,-178.461,5.822,148.574
C02421=1210.641,115.283,-50.148,-178.459,5.822,148.574
C02422=1210.636,115.533,-50.168,-178.456,5.824,148.573
C02423=1210.631,115.782,-50.188,-178.453,5.825,148.573
C02424=1210.626,116.031,-50.206,-178.451,5.826,148.572
C02425=1210.622,116.281,-50.226,-178.449,5.828,148.572
C02426=1210.616,116.529,-50.245,-178.446,5.828,148.571
C02427=1210.612,116.779,-50.265,-178.443,5.830,148.571
C02428=1210.608,117.028,-50.284,-178.441,5.831,148.570
C02429=1210.603,117.277,-50.304,-178.439,5.831,148.570
C02430=1210.598,117.526,-50.324,-178.435,5.833,148.569
C02431=1210.593,117.776,-50.343,-178.433,5.834,148.569
C02432=1210.588,118.025,-50.363,-178.430,5.835,148.568
C02433=1210.583,118.274,-50.382,-178.428,5.836,148.568
C02434=1210.578,118.523,-50.401,-178.425,5.837,148.567
C02435=1210.574,118.772,-50.421,-178.423,5.839,148.567
C02436=1210.569,119.022,-50.440,-178.420,5.839,148.566
C02437=1210.564,119.271,-50.460,-178.417,5.841,148.566
C02438=1210.559,119.520,-50.480,-178.415,5.842,148.565
C02439=1210.554,119.769,-50.500,-178.412,5.843,148.565
C02440=1210.550,120.018,-50.518,-178.410,5.844,148.564
C02441=1210.545,120.267,-50.538,-178.407,5.845,148.564
C02442=1210.540,120.517,-50.558,-178.404,5.846,148.563
C02443=1210.535,120.765,-50.578,-178.402,5.847,148.563
C02444=1210.530,121.015,-50.597,-178.399,5.849,148.562
C02445=1210.526,121.264,-50.617,-178.397,5.850,148.561
C02446=1210.521,121.514,-50.637,-178.394,5.851,148.561
C02447=1210.516,121.763,-50.656,-178.392,5.852,148.560
C02448=1210.511,122.012,-50.676,-178.389,5.853,148.560
C02449=1210.507,122.261,-50.695,-178.386,5.854,148.559
C02450=1210.502,122.510,-50.715,-178.384,5.855,148.559
C02451=1210.497,122.759,-50.734,-178.381,5.857,148.558
C02452=1210.493,123.008,-50.755,-178.379,5.858,148.558
C02453=1210.488,123.258,-50.774,-178.376,5.859,148.557
C02454=1210.483,123.507,-50.794,-178.374,5.860,148.557
C02455=1210.478,123.756,-50.814,-178.370,5.862,148.556
C02456=1210.473,124.005,-50.834,-178.368,5.863,148.556
C02457=1210.468,124.254,-50.853,-178.366,5.863,148.555
C02458=1210.464,124.503,-50.873,-178.363,5.865,148.555
C02459=1210.459,124.753,-50.893,-178.361,5.866,148.554
C02460=1210.454,125.002,-50.913,-178.358,5.867,148.554
C02461=1210.449,125.250,-50.933,-178.356,5.868,148.553
C02462=1210.444,125.500,-50.952,-178.352,5.870,148.553
C02463=1210.440,125.749,-50.973,-178.350,5.871,148.552
C02464=1210.435,125.999,-50.992,-178.347,5.872,148.552
C02465=1210.430,126.248,-51.012,-178.345,5.873,148.551
C02466=1210.425,126.496,-51.032,-178.342,5.875,148.551
C02467=1210.421,126.746,-51.052,-178.340,5.875,148.550
C02468=1210.416,126.995,-51.072,-178.338,5.876,148.550
C02469=1210.412,127.244,-51.092,-178.334,5.878,148.549
C02470=1210.407,127.493,-51.112,-178.332,5.879,148.549
C02471=1210.402,127.742,-51.131,-178.329,5.880,148.548
C02472=1210.397,127.991,-51.152,-178.327,5.881,148.548
C02473=1210.392,128.241,-51.172,-178.324,5.883,148.547
C02474=1210.387,128.490,-51.192,-178.322,5.884,148.547
C02475=1210.383,128.740,-51.212,-178.319,5.885,148.547
C02476=1210.378,128.988,-51.232,-178.316,5.886,148.546
C02477=1210.373,129.237,-51.252,-178.314,5.888,148.546
C02478=1210.368,129.486,-51.272,-178.311,5.888,148.545
C02479=1210.364,129.736,-51.292,-178.308,5.890,148.544
C02480=1210.359,129.985,-51.312,-178.306,5.891,148.544
C02481=1210.354,130.234,-51.332,-178.303,5.893,148.543
C02482=1210.349,130.483,-51.352,-178.301,5.894,148.543
C02483=1210.344,130.732,-51.373,-178.298,5.895,148.542
C02484=1210.340,130.982,-51.392,-178.296,5.896,148.542
C02485=1210.335,131.230,-51.413,-178.293,5.897,148.541
C02486=1210.330,131.480,-51.432,-178.290,5.898,148.541
C02487=1210.326,131.729,-51.453,-178.288,5.900,148.541
C02488=1210.321,131.978,-51.474,-178.285,5.901,148.540
C02489=1210.315,132.227,-51.493,-178.282,5.903,148.540
C02490=1210.311,132.476,-51.513,-178.280,5.903,148.539
C02491=1210.307,132.725,-51.534,-178.277,5.905,148.539
C02492=1210.301,132.994,-51.555,-178.275,5.906,148.538
C02493=1210.296,133.262,-51.577,-178.272,5.907,148.538
C02494=1210.291,133.532,-51.599,-178.269,5.909,148.537
C02495=1210.286,133.801,-51.621,-178.267,5.910,148.537
C02496=1210.281,134.050,-51.641,-178.263,5.911,148.536
C02497=1210.277,134.299,-51.662,-178.261,5.912,148.536
C02498=1210.272,134.547,-51.682,-178.258,5.914,148.535
C02499=1210.266,134.797,-51.702,-178.256,5.915,148.535
C02500=1210.262,135.046,-51.722,-178.253,5.916,148.534
C02501=1210.257,135.295,-51.743,-178.251,5.917,148.534
C02502=1210.253,135.544,-51.763,-178.248,5.919,148.533
C02503=1210.248,135.793,-51.784,-178.245,5.920,148.533
C02504=1210.243,136.042,-51.804,-178.243,5.921,148.532
C02505=1210.238,136.291,-51.824,-178.240,5.923,148.532
C02506=1210.233,136.541,-51.845,-178.238,5.924,148.531
C02507=1210.229,136.789,-51.865,-178.235,5.925,148.531
C02508=1210.224,137.038,-51.886,-178.233,5.926,148.530
C02509=1210.219,137.288,-51.906,-178.230,5.928,148.530
C02510=1210.215,137.537,-51.926,-178.227,5.929,148.529
C02511=1210.210,137.786,-51.947,-178.224,5.930,148.529
C02512=1210.205,138.035,-51.968,-178.222,5.931,148.528
C02513=1210.200,138.284,-51.988,-178.219,5.933,148.528
C02514=1210.196,138.533,-52.009,-178.217,5.934,148.527
C02515=1210.191,138.783,-52.030,-178.214,5.935,148.527
C02516=1210.186,139.032,-52.050,-178.212,5.936,148.526
C02517=1210.182,139.281,-52.070,-178.209,5.938,148.526
C02518=1210.177,139.530,-52.091,-178.206,5.940,148.526
C02519=1210.172,139.779,-52.111,-178.204,5.940,148.525
C02520=1210.167,140.029,-52.132,-178.201,5.942,148.524
C02521=1210.162,140.278,-52.152,-178.199,5.943,148.524
C02522=1210.158,140.527,-52.173,-178.196,5.944,148.523
C02523=1210.153,140.776,-52.194,-178.194,5.945,148.523
C02524=1210.148,141.025,-52.214,-178.191,5.947,148.523
C02525=1210.143,141.274,-52.235,-178.188,5.948,148.522
C02526=1210.139,141.523,-52.255,-178.186,5.949,148.522
C02527=1210.134,141.772,-52.276,-178.184,5.950,148.521
C02528=1210.129,142.021,-52.297,-178.180,5.952,148.521
C02529=1210.125,142.270,-52.317,-178.178,5.954,148.520
C02530=1210.120,142.519,-52.339,-178.176,5.955,148.520
C02531=1210.115,142.768,-52.359,-178.172,5.956,148.519
C02532=1210.110,143.017,-52.380,-178.170,5.957,148.519
C02533=1210.106,143.266,-52.400,-178.168,5.959,148.519
C02534=1210.101,143.515,-52.421,-178.165,5.960,148.518
C02535=1210.096,143.764,-52.442,-178.162,5.961,148.518
C02536=1210.091,144.013,-52.463,-178.160,5.963,148.517
C02537=1210.087,144.263,-52.483,-178.157,5.964,148.517
C02538=1210.082,144.512,-52.504,-178.154,5.966,148.516
C02539=1210.078,144.761,-52.525,-178.152,5.966,148.516
C02540=1210.073,145.010,-52.546,-178.149,5.968,148.515
C02541=1210.068,145.259,-52.567,-178.147,5.969,148.515
C02542=1210.063,145.508,-52.588,-178.144,5.971,148.514
C02543=1210.059,145.757,-52.608,-178.141,5.972,148.514
C02544=1210.054,146.006,-52.629,-178.139,5.973,148.513
C02545=1210.049,146.255,-52.651,-178.136,5.975,148.513
C02546=1210.045,146.505,-52.672,-178.134,5.976,148.512
C02547=1210.040,146.754,-52.693,-178.131,5.977,148.512
C02548=1210.035,147.003,-52.713,-178.128,5.979,148.512
C02549=1210.030,147.252,-52.734,-178.126,5.980,148.511
C02550=1210.025,147.501,-52.756,-178.123,5.982,148.511
C02551=1210.021,147.750,-52.776,-178.121,5.983,148.510
C02552=1210.016,147.999,-52.797,-178.118,5.984,148.510
C02553=1210.011,148.247,-52.818,-178.115,5.986,148.509
C02554=1210.007,148.497,-52.839,-178.113,5.987,148.509
C02555=1210.002,148.746,-52.860,-178.110,5.989,148.508
C02556=1209.997,148.995,-52.881,-178.108,5.989,148.508
C02557=1209.992,149.244,-52.902,-178.105,5.991,148.507
C02558=1209.987,149.493,-52.923,-178.102,5.993,148.507
C02559=1209.983,149.742,-52.944,-178.100,5.993,148.506
C02560=1209.978,149.992,-52.966,-178.097,5.995,148.506
C02561=1209.973,150.241,-52.987,-178.095,5.996,148.506
C02562=1209.969,150.489,-53.008,-178.092,5.998,148.505
C02563=1209.964,150.738,-53.029,-178.089,5.999,148.505
C02564=1209.959,150.988,-53.050,-178.087,6.000,148.504
C02565=1209.955,151.237,-53.071,-178.084,6.002,148.504
C02566=1209.950,151.486,-53.092,-178.082,6.003,148.503
C02567=1209.945,151.735,-53.114,-178.079,6.005,148.503
C02568=1209.940,151.984,-53.135,-178.077,6.006,148.503
C02569=1209.936,152.233,-53.155,-178.074,6.007,148.502
C02570=1209.931,152.482,-53.177,-178.071,6.009,148.502
C02571=1209.926,152.731,-53.198,-178.069,6.011,148.501
C02572=1209.921,152.980,-53.220,-178.066,6.012,148.501
C02573=1209.917,153.229,-53.240,-178.063,6.013,148.500
C02574=1209.913,153.478,-53.262,-178.061,6.014,148.500
C02575=1209.907,153.728,-53.283,-178.059,6.016,148.499
C02576=1209.903,153.976,-53.305,-178.055,6.017,148.499
C02577=1209.898,154.225,-53.325,-178.053,6.018,148.498
C02578=1209.894,154.475,-53.347,-178.051,6.020,148.498
C02579=1209.889,154.724,-53.368,-178.048,6.022,148.498
C02580=1209.884,154.972,-53.390,-178.045,6.022,148.497
C02581=1209.879,155.221,-53.412,-178.043,6.024,148.497
C02582=1209.875,155.471,-53.432,-178.040,6.026,148.496
C02583=1209.870,155.719,-53.454,-178.038,6.027,148.496
C02584=1209.865,155.969,-53.475,-178.035,6.029,148.495
C02585=1209.861,156.218,-53.497,-178.033,6.029,148.495
C02586=1209.856,156.467,-53.519,-178.030,6.031,148.495
C02587=1209.851,156.716,-53.540,-178.027,6.033,148.494
C02588=1209.846,156.965,-53.561,-178.025,6.034,148.494
C02589=1209.842,157.214,-53.582,-178.022,6.036,148.493
C02590=1209.837,157.463,-53.604,-178.019,6.037,148.493
C02591=1209.832,157.711,-53.626,-178.017,6.038,148.492
C02592=1209.828,157.961,-53.647,-178.014,6.040,148.492
C02593=1209.823,158.210,-53.669,-178.011,6.042,148.491
C02594=1209.818,158.459,-53.690,-178.009,6.043,148.491
C02595=1209.814,158.708,-53.712,-178.006,6.044,148.490
C02596=1209.809,158.977,-53.735,-178.004,6.046,148.490
C02597=1209.803,159.246,-53.758,-178.001,6.048,148.490
C02598=1209.799,159.515,-53.782,-177.998,6.049,148.489
C02599=1209.794,159.784,-53.805,-177.995,6.051,148.489
C02600=1209.789,160.033,-53.827,-177.993,6.052,148.488
C02601=1209.784,160.282,-53.848,-177.990,6.053,148.488
C02602=1209.779,160.531,-53.870,-177.987,6.055,148.487
C02603=1209.774,160.780,-53.892,-177.985,6.056,148.487
C02604=1209.770,161.029,-53.913,-177.982,6.058,148.487
C02605=1209.765,161.278,-53.935,-177.979,6.059,148.486
C02606=1209.760,161.527,-53.956,-177.977,6.060,148.486
C02607=1209.756,161.777,-53.978,-177.974,6.062,148.485
C02608=1209.751,162.025,-54.000,-177.972,6.064,148.485
C02609=1209.746,162.274,-54.022,-177.969,6.065,148.484
C02610=1209.742,162.523,-54.044,-177.966,6.066,148.484
C02611=1209.737,162.772,-54.065,-177.964,6.068,148.484
C02612=1209.733,163.021,-54.087,-177.962,6.069,148.483
C02613=1209.727,163.271,-54.108,-177.959,6.071,148.483
C02614=1209.723,163.520,-54.131,-177.956,6.072,148.482
C02615=1209.718,163.769,-54.152,-177.953,6.074,148.482
C02616=1209.713,164.017,-54.174,-177.951,6.075,148.481
C02617=1209.709,164.267,-54.196,-177.948,6.077,148.481
C02618=1209.704,164.515,-54.218,-177.946,6.079,148.481
C02619=1209.700,164.765,-54.240,-177.943,6.079,148.480
C02620=1209.695,165.013,-54.261,-177.941,6.081,148.480
C02621=1209.691,165.262,-54.283,-177.938,6.083,148.479
C02622=1209.686,165.511,-54.305,-177.935,6.085,148.479
C02623=1209.680,165.760,-54.327,-177.933,6.086,148.479
C02624=1209.676,166.009,-54.349,-177.930,6.087,148.478
C02625=1209.671,166.258,-54.371,-177.927,6.089,148.478
C02626=1209.667,166.507,-54.393,-177.925,6.090,148.477
C02627=1209.662,166.756,-54.415,-177.923,6.092,148.477
C02628=1209.658,167.005,-54.437,-177.920,6.094,148.477
C02629=1209.653,167.254,-54.459,-177.917,6.095,148.476
C02630=1209.648,167.504,-54.481,-177.915,6.096,148.476
C02631=1209.643,167.752,-54.503,-177.912,6.098,148.475
C02632=1209.639,168.002,-54.525,-177.909,6.100,148.475
C02633=1209.634,168.250,-54.547,-177.907,6.101,148.474
C02634=1209.630,168.499,-54.569,-177.904,6.102,148.474
C02635=1209.625,168.748,-54.591,-177.901,6.104,148.474
C02636=1209.620,168.997,-54.614,-177.899,6.106,148.473
C02637=1209.615,169.246,-54.635,-177.897,6.107,148.473
C02638=1209.611,169.495,-54.657,-177.894,6.109,148.472
C02639=1209.606,169.744,-54.679,-177.891,6.110,148.472
C02640=1209.602,169.993,-54.702,-177.888,6.112,148.471
C02641=1209.597,170.242,-54.724,-177.886,6.113,148.471
C02642=1209.592,170.491,-54.746,-177.883,6.115,148.471
C02643=1209.588,170.740,-54.768,-177.881,6.117,148.470
C02644=1209.583,170.989,-54.790,-177.878,6.118,148.470
C02645=1209.579,171.238,-54.813,-177.875,6.119,148.469
C02646=1209.574,171.487,-54.835,-177.873,6.121,148.469
C02647=1209.569,171.736,-54.857,-177.870,6.123,148.469
C02648=1209.564,171.985,-54.879,-177.867,6.124,148.468
C02649=1209.560,172.234,-54.902,-177.865,6.125,148.468
C02650=1209.555,172.482,-54.924,-177.863,6.127,148.468
C02651=1209.551,172.732,-54.946,-177.860,6.129,148.467
C02652=1209.546,172.981,-54.969,-177.857,6.131,148.467
C02653=1209.541,173.229,-54.991,-177.855,6.132,148.466
C02654=1209.537,173.479,-55.013,-177.852,6.133,148.466
C02655=1209.531,173.728,-55.035,-177.849,6.135,148.465
C02656=1209.527,173.976,-55.058,-177.847,6.137,148.465
C02657=1209.523,174.226,-55.080,-177.845,6.138,148.465
C02658=1209.518,174.474,-55.103,-177.842,6.139,148.464
C02659=1209.513,174.723,-55.125,-177.839,6.141,148.464
C02660=1209.508,174.972,-55.147,-177.836,6.143,148.463
C02661=1209.504,175.221,-55.170,-177.834,6.144,148.463
C02662=1209.500,175.470,-55.192,-177.831,6.146,148.463
C02663=1209.494,175.719,-55.215,-177.829,6.148,148.462
C02664=1209.490,175.968,-55.237,-177.826,6.149,148.462
C02665=1209.485,176.218,-55.260,-177.823,6.151,148.461
C02666=1209.480,176.466,-55.282,-177.821,6.152,148.461
C02667=1209.476,176.715,-55.304,-177.818,6.154,148.461
C02668=1209.471,176.964,-55.328,-177.816,6.156,148.460
C02669=1209.467,177.213,-55.349,-177.813,6.157,148.460
C02670=1209.462,177.462,-55.373,-177.811,6.158,148.460
C02671=1209.458,177.711,-55.395,-177.808,6.160,148.459
C02672=1209.452,177.959,-55.418,-177.806,6.162,148.459
C02673=1209.448,178.209,-55.440,-177.802,6.163,148.458
C02674=1209.444,178.457,-55.462,-177.800,6.165,148.458
C02675=1209.439,178.706,-55.485,-177.798,6.166,148.457
C02676=1209.435,178.955,-55.508,-177.795,6.168,148.457
C02677=1209.430,179.205,-55.530,-177.792,6.170,148.457
C02678=1209.425,179.453,-55.553,-177.790,6.172,148.456
C02679=1209.420,179.702,-55.576,-177.787,6.174,148.456
C02680=1209.416,179.951,-55.598,-177.785,6.175,148.456
C02681=1209.411,180.200,-55.621,-177.782,6.176,148.455
C02682=1209.406,180.449,-55.643,-177.779,6.178,148.455
C02683=1209.402,180.698,-55.666,-177.776,6.180,148.454
C02684=1209.398,180.947,-55.689,-177.774,6.181,148.454
C02685=1209.392,181.196,-55.711,-177.772,6.182,148.454
C02686=1209.387,181.445,-55.735,-177.769,6.184,148.453
C02687=1209.384,181.693,-55.758,-177.766,6.186,148.453
C02688=1209.379,181.943,-55.780,-177.764,6.188,148.453
C02689=1209.374,182.191,-55.803,-177.761,6.190,148.452
C02690=1209.369,182.440,-55.826,-177.758,6.192,148.452
C02691=1209.365,182.689,-55.848,-177.756,6.193,148.451
C02692=1209.360,182.938,-55.871,-177.753,6.194,148.451
C02693=1209.356,183.187,-55.895,-177.751,6.196,148.451
C02694=1209.351,183.435,-55.917,-177.748,6.198,148.450
C02695=1209.346,183.685,-55.940,-177.745,6.199,148.450
C02696=1209.342,183.934,-55.962,-177.743,6.201,148.450
C02697=1209.337,184.183,-55.986,-177.740,6.202,148.449
C02698=1209.332,184.431,-56.009,-177.738,6.204,148.449
C02699=1209.328,184.680,-56.032,-177.735,6.206,148.448
C02700=1209.323,184.950,-56.057,-177.732,6.208,148.448
C02701=1209.317,185.219,-56.082,-177.729,6.209,148.447
C02702=1209.313,185.489,-56.106,-177.727,6.211,148.447
C02703=1209.308,185.759,-56.131,-177.724,6.213,148.447
C02704=1209.303,186.008,-56.155,-177.721,6.215,148.446
C02705=1209.299,186.256,-56.177,-177.719,6.216,148.446
C02706=1209.294,186.506,-56.200,-177.716,6.218,148.446
C02707=1209.289,186.755,-56.223,-177.713,6.220,148.445
C02708=1209.285,187.003,-56.246,-177.710,6.222,148.445
C02709=1209.280,187.252,-56.269,-177.708,6.223,148.444
C02710=1209.275,187.501,-56.292,-177.706,6.224,148.444
C02711=1209.271,187.750,-56.315,-177.703,6.226,148.444
C02712=1209.267,187.999,-56.339,-177.700,6.228,148.443
C02713=1209.262,188.248,-56.362,-177.698,6.230,148.443
C02714=1209.257,188.497,-56.385,-177.695,6.232,148.443
C02715=1209.253,188.745,-56.408,-177.692,6.234,148.442
C02716=1209.248,188.994,-56.431,-177.690,6.235,148.442
C02717=1209.243,189.243,-56.454,-177.688,6.236,148.442
C02718=1209.239,189.492,-56.478,-177.685,6.238,148.441
C02719=1209.234,189.741,-56.501,-177.682,6.240,148.441
C02720=1209.230,189.990,-56.524,-177.680,6.242,148.441
C02721=1209.225,190.239,-56.547,-177.677,6.244,148.440
C02722=1209.220,190.488,-56.571,-177.674,6.245,148.440
C02723=1209.216,190.737,-56.594,-177.672,6.247,148.439
C02724=1209.210,190.985,-56.617,-177.670,6.248,148.439
C02725=1209.206,191.234,-56.640,-177.667,6.250,148.439
C02726=1209.202,191.483,-56.663,-177.664,6.252,148.438
C02727=1209.197,191.732,-56.686,-177.662,6.254,148.438
C02728=1209.192,191.981,-56.710,-177.659,6.256,148.438
C02729=1209.188,192.230,-56.733,-177.656,6.257,148.437
C02730=1209.183,192.479,-56.757,-177.653,6.259,148.437
C02731=1209.179,192.728,-56.781,-177.650,6.261,148.436
C02732=1209.174,192.977,-56.804,-177.648,6.262,148.436
C02733=1209.169,193.226,-56.827,-177.646,6.264,148.436
C02734=1209.165,193.474,-56.850,-177.643,6.265,148.435
C02735=1209.161,193.723,-56.873,-177.640,6.267,148.435
C02736=1209.156,193.972,-56.897,-177.638,6.269,148.435
C02737=1209.151,194.221,-56.921,-177.635,6.271,148.434
C02738=1209.147,194.470,-56.944,-177.632,6.273,148.434
C02739=1209.142,194.719,-56.968,-177.630,6.274,148.434
C02740=1209.138,194.967,-56.992,-177.627,6.276,148.433
C02741=1209.132,195.216,-57.015,-177.625,6.278,148.433
C02742=1209.128,195.465,-57.038,-177.622,6.279,148.433
C02743=1209.123,195.714,-57.061,-177.620,6.281,148.432
C02744=1209.119,195.962,-57.085,-177.617,6.283,148.432
C02745=1209.114,196.211,-57.109,-177.614,6.285,148.432
C02746=1209.109,196.460,-57.132,-177.612,6.286,148.431
C02747=1209.104,196.709,-57.155,-177.609,6.288,148.431
C02748=1209.101,196.958,-57.180,-177.607,6.290,148.430
C02749=1209.096,197.207,-57.203,-177.604,6.292,148.430
C02750=1209.091,197.456,-57.227,-177.601,6.294,148.430
C02751=1209.087,197.705,-57.251,-177.599,6.296,148.429
C02752=1209.082,197.954,-57.274,-177.596,6.297,148.429
C02753=1209.078,198.202,-57.298,-177.593,6.299,148.429
C02754=1209.073,198.451,-57.321,-177.591,6.301,148.428
C02755=1209.068,198.700,-57.345,-177.589,6.302,148.428
C02756=1209.064,198.949,-57.369,-177.586,6.304,148.428
C02757=1209.059,199.198,-57.392,-177.583,6.306,148.427
C02758=1209.055,199.446,-57.416,-177.581,6.308,148.427
C02759=1209.050,199.695,-57.440,-177.578,6.309,148.427
C02760=1209.046,199.944,-57.464,-177.575,6.311,148.426
C02761=1209.041,200.193,-57.487,-177.573,6.313,148.426
C02762=1209.036,200.441,-57.512,-177.570,6.315,148.426
C02763=1209.031,200.690,-57.535,-177.567,6.317,148.425
C02764=1209.027,200.939,-57.559,-177.565,6.318,148.425
C02765=1209.022,201.188,-57.583,-177.563,6.321,148.425
C02766=1209.018,201.437,-57.607,-177.560,6.322,148.424
C02767=1209.014,201.686,-57.630,-177.557,6.324,148.424
C02768=1209.009,201.934,-57.654,-177.555,6.326,148.424
C02769=1209.005,202.183,-57.678,-177.552,6.328,148.423
C02770=1208.999,202.432,-57.703,-177.549,6.330,148.423
C02771=1208.995,202.681,-57.726,-177.547,6.332,148.423
C02772=1208.990,202.930,-57.750,-177.545,6.333,148.422
C02773=1208.986,203.179,-57.773,-177.542,6.334,148.422
C02774=1208.982,203.428,-57.798,-177.539,6.336,148.422
C02775=1208.977,203.676,-57.822,-177.537,6.338,148.421
C02776=1208.972,203.925,-57.846,-177.534,6.340,148.421
C02777=1208.968,204.174,-57.870,-177.531,6.342,148.421
C02778=1208.963,204.422,-57.894,-177.529,6.344,148.420
C02779=1208.959,204.671,-57.917,-177.526,6.345,148.420
C02780=1208.953,204.920,-57.942,-177.523,6.347,148.420
C02781=1208.950,205.169,-57.966,-177.521,6.349,148.419
C02782=1208.945,205.418,-57.990,-177.518,6.351,148.419
C02783=1208.941,205.667,-58.014,-177.515,6.353,148.419
C02784=1208.935,205.915,-58.038,-177.513,6.355,148.418
C02785=1208.931,206.164,-58.063,-177.510,6.356,148.418
C02786=1208.927,206.414,-58.086,-177.508,6.358,148.418
C02787=1208.922,206.662,-58.110,-177.505,6.360,148.418
C02788=1208.917,206.911,-58.135,-177.503,6.362,148.417
C02789=1208.913,207.159,-58.159,-177.500,6.364,148.417
C02790=1208.908,207.408,-58.182,-177.497,6.366,148.417
C02791=1208.904,207.658,-58.207,-177.495,6.368,148.416
C02792=1208.899,207.906,-58.232,-177.492,6.370,148.416
C02793=1208.895,208.154,-58.256,-177.489,6.371,148.416
C02794=1208.890,208.403,-58.280,-177.487,6.373,148.415
C02795=1208.885,208.652,-58.304,-177.484,6.375,148.415
C02796=1208.881,208.901,-58.328,-177.482,6.377,148.414
C02797=1208.876,209.150,-58.353,-177.479,6.379,148.414
C02798=1208.872,209.398,-58.377,-177.476,6.381,148.414
C02799=1208.867,209.647,-58.401,-177.474,6.382,148.413
C02800=1208.863,209.896,-58.426,-177.471,6.385,148.413
C02801=1208.858,210.145,-58.450,-177.469,6.386,148.413
C02802=1208.853,210.393,-58.475,-177.466,6.388,148.413
C02803=1208.849,210.642,-58.499,-177.464,6.390,148.412
C02804=1208.844,210.913,-58.525,-177.461,6.392,148.412
C02805=1208.839,211.183,-58.552,-177.458,6.395,148.412
C02806=1208.835,211.453,-58.578,-177.455,6.396,148.411
C02807=1208.829,211.723,-58.605,-177.452,6.398,148.411
C02808=1208.825,211.973,-58.630,-177.450,6.400,148.411
C02809=1208.820,212.221,-58.654,-177.447,6.402,148.410
C02810=1208.815,212.470,-58.678,-177.444,6.404,148.410
C02811=1208.811,212.718,-58.703,-177.442,6.406,148.410
C02812=1208.806,212.968,-58.728,-177.439,6.407,148.409
C02813=1208.802,213.216,-58.752,-177.437,6.409,148.409
C02814=1208.797,213.465,-58.776,-177.434,6.411,148.409
C02815=1208.793,213.714,-58.801,-177.431,6.413,148.408
C02816=1208.788,213.963,-58.825,-177.429,6.415,148.408
C02817=1208.784,214.211,-58.850,-177.426,6.417,148.408
C02818=1208.779,214.461,-58.875,-177.424,6.419,148.408
C02819=1208.775,214.709,-58.899,-177.421,6.421,148.407
C02820=1208.769,214.958,-58.923,-177.419,6.422,148.407
C02821=1208.766,215.207,-58.948,-177.415,6.425,148.407
C02822=1208.761,215.455,-58.973,-177.413,6.427,148.406
C02823=1208.756,215.703,-58.997,-177.410,6.429,148.406
C02824=1208.752,215.953,-59.022,-177.407,6.431,148.406
C02825=1208.748,216.201,-59.046,-177.405,6.433,148.406
C02826=1208.743,216.451,-59.071,-177.403,6.435,148.405
C02827=1208.738,216.699,-59.096,-177.400,6.436,148.405
C02828=1208.734,216.947,-59.121,-177.397,6.438,148.405
C02829=1208.729,217.197,-59.146,-177.395,6.440,148.404
C02830=1208.725,217.445,-59.170,-177.392,6.442,148.404
C02831=1208.720,217.694,-59.195,-177.389,6.444,148.404
C02832=1208.716,217.943,-59.220,-177.387,6.446,148.403
C02833=1208.711,218.191,-59.244,-177.385,6.448,148.403
C02834=1208.707,218.440,-59.269,-177.382,6.450,148.403
C02835=1208.702,218.689,-59.294,-177.379,6.452,148.402
C02836=1208.698,218.938,-59.319,-177.377,6.453,148.402
C02837=1208.693,219.186,-59.344,-177.374,6.455,148.402
C02838=1208.688,219.435,-59.368,-177.371,6.457,148.401
C02839=1208.684,219.684,-59.394,-177.369,6.459,148.401
C02840=1208.679,219.932,-59.418,-177.366,6.462,148.401
C02841=1208.675,220.181,-59.443,-177.363,6.464,148.401
C02842=1208.670,220.429,-59.468,-177.361,6.466,148.400
C02843=1208.666,220.679,-59.493,-177.358,6.467,148.400
C02844=1208.661,220.927,-59.519,-177.356,6.469,148.400
C02845=1208.657,221.176,-59.543,-177.353,6.471,148.400
C02846=1208.652,221.425,-59.568,-177.351,6.473,148.399
C02847=1208.648,221.674,-59.594,-177.348,6.475,148.399
C02848=1208.644,221.922,-59.618,-177.345,6.477,148.399
C02849=1208.639,222.171,-59.643,-177.343,6.479,148.398
C02850=1208.634,222.420,-59.668,-177.341,6.481,148.398
C02851=1208.630,222.668,-59.694,-177.338,6.483,148.398
C02852=1208.625,222.917,-59.718,-177.335,6.485,148.398
C02853=1208.621,223.166,-59.744,-177.333,6.486,148.397
C02854=1208.616,223.414,-59.768,-177.330,6.488,148.397
C02855=1208.612,223.663,-59.794,-177.327,6.491,148.397
C02856=1208.607,223.912,-59.819,-177.325,6.493,148.396
C02857=1208.603,224.160,-59.844,-177.322,6.495,148.396
C02858=1208.598,224.409,-59.869,-177.320,6.497,148.396
C02859=1208.594,224.658,-59.894,-177.317,6.499,148.395
C02860=1208.589,224.907,-59.919,-177.314,6.501,148.395
C02861=1208.585,225.155,-59.945,-177.312,6.503,148.395
C02862=1208.580,225.404,-59.969,-177.309,6.505,148.395
C02863=1208.576,225.653,-59.995,-177.307,6.506,148.394
C02864=1208.571,225.901,-60.020,-177.304,6.508,148.394
C02865=1208.567,226.150,-60.045,-177.302,6.510,148.394
C02866=1208.562,226.398,-60.070,-177.299,6.513,148.394
C02867=1208.558,226.647,-60.096,-177.296,6.515,148.393
C02868=1208.553,226.896,-60.121,-177.294,6.517,148.393
C02869=1208.548,227.145,-60.146,-177.291,6.519,148.393
C02870=1208.544,227.393,-60.172,-177.289,6.521,148.393
C02871=1208.539,227.642,-60.197,-177.286,6.523,148.392
C02872=1208.535,227.891,-60.222,-177.284,6.524,148.392
C02873=1208.531,228.139,-60.247,-177.281,6.526,148.392
C02874=1208.526,228.388,-60.272,-177.279,6.528,148.391
C02875=1208.522,228.637,-60.298,-177.276,6.530,148.391
C02876=1208.517,228.885,-60.324,-177.273,6.532,148.391
C02877=1208.513,229.134,-60.349,-177.270,6.535,148.391
C02878=1208.508,229.383,-60.374,-177.268,6.537,148.390
C02879=1208.503,229.631,-60.400,-177.265,6.539,148.390
C02880=1208.499,229.880,-60.426,-177.263,6.541,148.390
C02881=1208.494,230.128,-60.451,-177.260,6.543,148.389
C02882=1208.490,230.377,-60.477,-177.258,6.545,148.389
C02883=1208.486,230.626,-60.502,-177.255,6.547,148.389
C02884=1208.481,230.875,-60.527,-177.253,6.548,148.389
C02885=1208.477,231.123,-60.553,-177.250,6.550,148.388
C02886=1208.472,231.372,-60.579,-177.247,6.553,148.388
C02887=1208.468,231.620,-60.604,-177.245,6.555,148.388
C02888=1208.463,231.869,-60.630,-177.242,6.557,148.388
C02889=1208.459,232.117,-60.655,-177.240,6.559,148.387
C02890=1208.454,232.366,-60.681,-177.237,6.561,148.387
C02891=1208.450,232.615,-60.707,-177.235,6.563,148.387
C02892=1208.445,232.864,-60.731,-177.232,6.565,148.387
C02893=1208.440,233.113,-60.758,-177.230,6.567,148.386
C02894=1208.436,233.361,-60.783,-177.227,6.570,148.386
C02895=1208.432,233.610,-60.809,-177.224,6.571,148.386
C02896=1208.427,233.858,-60.835,-177.222,6.573,148.386
C02897=1208.422,234.107,-60.860,-177.219,6.575,148.386
C02898=1208.418,234.356,-60.886,-177.217,6.577,148.385
C02899=1208.413,234.604,-60.911,-177.214,6.579,148.385
C02900=1208.409,234.853,-60.937,-177.212,6.581,148.385
C02901=1208.405,235.102,-60.963,-177.209,6.584,148.384
C02902=1208.400,235.351,-60.989,-177.206,6.586,148.384
C02903=1208.395,235.599,-61.015,-177.204,6.588,148.384
C02904=1208.391,235.848,-61.040,-177.201,6.590,148.384
C02905=1208.387,236.096,-61.067,-177.199,6.592,148.383
C02906=1208.382,236.344,-61.092,-177.196,6.594,148.383
C02907=1208.378,236.593,-61.118,-177.193,6.595,148.383
C02908=1208.373,236.865,-61.147,-177.191,6.598,148.383
C02909=1208.367,237.136,-61.174,-177.188,6.600,148.382
C02910=1208.363,237.408,-61.203,-177.185,6.603,148.382
C02911=1208.358,237.679,-61.231,-177.182,6.605,148.382
C02912=1208.354,237.928,-61.257,-177.180,6.607,148.381
C02913=1208.349,238.176,-61.283,-177.178,6.609,148.381
C02914=1208.344,238.425,-61.309,-177.174,6.611,148.381
C02915=1208.340,238.674,-61.335,-177.172,6.613,148.381
C02916=1208.336,238.922,-61.361,-177.170,6.615,148.381
C02917=1208.331,239.171,-61.386,-177.167,6.617,148.380
C02918=1208.327,239.419,-61.413,-177.164,6.619,148.380
C02919=1208.322,239.668,-61.439,-177.162,6.621,148.380
C02920=1208.318,239.917,-61.465,-177.159,6.624,148.380
C02921=1208.314,240.165,-61.490,-177.156,6.626,148.379
C02922=1208.309,240.413,-61.517,-177.154,6.628,148.379
C02923=1208.304,240.662,-61.543,-177.152,6.630,148.379
C02924=1208.300,240.911,-61.569,-177.149,6.632,148.379
C02925=1208.296,241.159,-61.596,-177.147,6.634,148.379
C02926=1208.291,241.408,-61.622,-177.144,6.637,148.378
C02927=1208.287,241.657,-61.647,-177.141,6.638,148.378
C02928=1208.282,241.905,-61.674,-177.139,6.641,148.378
C02929=1208.278,242.154,-61.700,-177.136,6.643,148.378
C02930=1208.273,242.402,-61.725,-177.134,6.644,148.377
C02931=1208.269,242.651,-61.753,-177.131,6.647,148.377
C02932=1208.264,242.900,-61.778,-177.128,6.649,148.377
C02933=1208.260,243.149,-61.805,-177.126,6.651,148.377
C02934=1208.256,243.397,-61.831,-177.123,6.653,148.376
C02935=1208.251,243.646,-61.857,-177.121,6.655,148.376
C02936=1208.246,243.894,-61.884,-177.118,6.658,148.376
C02937=1208.242,244.142,-61.909,-177.116,6.660,148.376
C02938=1208.237,244.391,-61.936,-177.113,6.662,148.375
C02939=1208.233,244.640,-61.962,-177.111,6.664,148.375
C02940=1208.229,244.888,-61.989,-177.108,6.666,148.375
C02941=1208.224,245.137,-62.015,-177.105,6.669,148.375
C02942=1208.220,245.385,-62.041,-177.103,6.671,148.375
C02943=1208.215,245.634,-62.068,-177.100,6.673,148.374
C02944=1208.211,245.882,-62.094,-177.098,6.675,148.374
C02945=1208.206,246.132,-62.121,-177.095,6.677,148.374
C02946=1208.202,246.379,-62.147,-177.092,6.679,148.374
C02947=1208.197,246.628,-62.173,-177.090,6.681,148.374
C02948=1208.193,246.876,-62.199,-177.087,6.683,148.373
C02949=1208.188,247.125,-62.226,-177.085,6.686,148.373
C02950=1208.184,247.374,-62.252,-177.083,6.687,148.373
C02951=1208.179,247.622,-62.279,-177.080,6.690,148.373
C02952=1208.175,247.871,-62.305,-177.077,6.692,148.372
C02953=1208.171,248.119,-62.332,-177.075,6.694,148.372
C02954=1208.166,248.368,-62.358,-177.073,6.696,148.372
C02955=1208.162,248.617,-62.385,-177.069,6.699,148.372
C02956=1208.158,248.865,-62.411,-177.067,6.701,148.371
C02957=1208.153,249.114,-62.438,-177.065,6.703,148.371
C02958=1208.148,249.363,-62.465,-177.062,6.705,148.371
C02959=1208.144,249.611,-62.491,-177.060,6.707,148.371
C02960=1208.140,249.859,-62.518,-177.057,6.710,148.371
C02961=1208.135,250.108,-62.544,-177.054,6.712,148.370
C02962=1208.131,250.357,-62.571,-177.052,6.714,148.370
C02963=1208.127,250.605,-62.598,-177.049,6.716,148.370
C02964=1208.122,250.853,-62.625,-177.047,6.719,148.370
C02965=1208.117,251.102,-62.651,-177.044,6.720,148.370
C02966=1208.113,251.350,-62.677,-177.042,6.723,148.370
C02967=1208.109,251.599,-62.705,-177.039,6.725,148.369
C02968=1208.104,251.847,-62.732,-177.036,6.727,148.369
C02969=1208.100,252.096,-62.757,-177.034,6.729,148.369
C02970=1208.095,252.345,-62.784,-177.031,6.731,148.369
C02971=1208.090,252.593,-62.811,-177.029,6.733,148.368
C02972=1208.086,252.841,-62.838,-177.026,6.736,148.368
C02973=1208.082,253.090,-62.865,-177.024,6.738,148.368
C02974=1208.077,253.338,-62.892,-177.021,6.740,148.368
C02975=1208.073,253.587,-62.919,-177.019,6.742,148.368
C02976=1208.069,253.835,-62.946,-177.016,6.745,148.367
C02977=1208.064,254.085,-62.972,-177.014,6.747,148.367
C02978=1208.060,254.333,-62.999,-177.011,6.749,148.367
C02979=1208.056,254.582,-63.026,-177.008,6.751,148.367
C02980=1208.051,254.830,-63.053,-177.006,6.754,148.367
C02981=1208.046,255.079,-63.080,-177.003,6.756,148.366
C02982=1208.042,255.327,-63.106,-177.001,6.758,148.366
C02983=1208.038,255.575,-63.133,-176.998,6.760,148.366
C02984=1208.033,255.824,-63.161,-176.996,6.763,148.366
C02985=1208.028,256.072,-63.188,-176.993,6.765,148.366
C02986=1208.024,256.321,-63.215,-176.991,6.767,148.366
C02987=1208.020,256.570,-63.242,-176.988,6.770,148.365
C02988=1208.016,256.818,-63.269,-176.986,6.772,148.365
C02989=1208.011,257.067,-63.296,-176.983,6.774,148.365
C02990=1208.006,257.315,-63.323,-176.981,6.776,148.365
C02991=1208.002,257.564,-63.350,-176.978,6.779,148.365
C02992=1207.998,257.812,-63.376,-176.976,6.781,148.364
C02993=1207.994,258.060,-63.404,-176.973,6.783,148.364
C02994=1207.989,258.309,-63.431,-176.970,6.786,148.364
C02995=1207.985,258.557,-63.458,-176.968,6.787,148.364
C02996=1207.980,258.806,-63.486,-176.965,6.790,148.364
C02997=1207.976,259.054,-63.513,-176.963,6.791,148.363
C02998=1207.971,259.303,-63.540,-176.960,6.794,148.363
C02999=1207.967,259.551,-63.566,-176.957,6.796,148.363
C03000=1207.963,259.800,-63.594,-176.955,6.799,148.363
C03001=1207.959,260.048,-63.621,-176.952,6.801,148.363
C03002=1207.954,260.297,-63.648,-176.950,6.803,148.363
C03003=1207.949,260.545,-63.675,-176.947,6.805,148.362
C03004=1207.945,260.794,-63.703,-176.945,6.808,148.362
C03005=1207.940,261.042,-63.730,-176.942,6.810,148.362
C03006=1207.936,261.291,-63.758,-176.940,6.812,148.362
C03007=1207.931,261.539,-63.785,-176.937,6.815,148.362
C03008=1207.927,261.788,-63.812,-176.935,6.817,148.362
C03009=1207.922,262.036,-63.840,-176.932,6.819,148.361
C03010=1207.918,262.285,-63.867,-176.930,6.821,148.361
C03011=1207.914,262.533,-63.894,-176.927,6.824,148.361
C03012=1207.909,262.806,-63.924,-176.925,6.826,148.361
C03013=1207.904,263.078,-63.954,-176.921,6.829,148.361
C03014=1207.900,263.351,-63.984,-176.919,6.832,148.361
C03015=1207.895,263.624,-64.015,-176.916,6.834,148.360
C03016=1207.890,263.872,-64.042,-176.913,6.836,148.360
C03017=1207.886,264.120,-64.069,-176.911,6.839,148.360
C03018=1207.882,264.369,-64.097,-176.909,6.841,148.360
C03019=1207.877,264.618,-64.124,-176.905,6.843,148.360
C03020=1207.873,264.866,-64.152,-176.903,6.846,148.359
C03021=1207.868,265.114,-64.179,-176.901,6.848,148.359
C03022=1207.864,265.363,-64.207,-176.898,6.851,148.359
C03023=1207.860,265.611,-64.234,-176.895,6.852,148.359
C03024=1207.855,265.860,-64.261,-176.893,6.855,148.359
C03025=1207.851,266.109,-64.290,-176.890,6.857,148.358
C03026=1207.846,266.357,-64.317,-176.888,6.859,148.358
C03027=1207.842,266.605,-64.345,-176.886,6.862,148.358
C03028=1207.837,266.854,-64.372,-176.883,6.864,148.358
C03029=1207.833,267.102,-64.400,-176.880,6.867,148.358
C03030=1207.829,267.350,-64.428,-176.878,6.868,148.358
C03031=1207.824,267.599,-64.455,-176.875,6.871,148.358
C03032=1207.820,267.847,-64.483,-176.873,6.873,148.357
C03033=1207.815,268.096,-64.510,-176.870,6.876,148.357
C03034=1207.811,268.344,-64.538,-176.868,6.878,148.357
C03035=1207.807,268.593,-64.566,-176.865,6.880,148.357
C03036=1207.802,268.841,-64.593,-176.862,6.883,148.357
C03037=1207.798,269.089,-64.621,-176.860,6.885,148.357
C03038=1207.794,269.338,-64.649,-176.858,6.887,148.357
C03039=1207.789,269.586,-64.677,-176.855,6.890,148.356
C03040=1207.785,269.835,-64.704,-176.852,6.892,148.356
C03041=1207.780,270.083,-64.732,-176.850,6.895,148.356
C03042=1207.776,270.331,-64.760,-176.847,6.897,148.356
C03043=1207.771,270.580,-64.789,-176.845,6.899,148.356
C03044=1207.767,270.828,-64.816,-176.842,6.902,148.356
C03045=1207.762,271.076,-64.844,-176.840,6.904,148.355
C03046=1207.759,271.325,-64.872,-176.837,6.906,148.355
C03047=1207.754,271.573,-64.899,-176.835,6.909,148.355
C03048=1207.750,271.822,-64.927,-176.832,6.911,148.355
C03049=1207.745,272.070,-64.955,-176.829,6.914,148.355
C03050=1207.741,272.319,-64.983,-176.827,6.916,148.355
C03051=1207.736,272.568,-65.011,-176.825,6.918,148.355
C03052=1207.732,272.815,-65.039,-176.822,6.921,148.355
C03053=1207.728,273.064,-65.067,-176.819,6.923,148.354
C03054=1207.723,273.312,-65.095,-176.817,6.926,148.354
C03055=1207.719,273.561,-65.123,-176.815,6.929,148.354
C03056=1207.715,273.809,-65.151,-176.812,6.930,148.354
C03057=1207.710,274.058,-65.179,-176.809,6.933,148.354
C03058=1207.706,274.306,-65.207,-176.807,6.936,148.354
C03059=1207.701,274.554,-65.235,-176.805,6.937,148.353
C03060=1207.697,274.803,-65.264,-176.802,6.940,148.353
C03061=1207.692,275.051,-65.291,-176.800,6.943,148.353
C03062=1207.689,275.299,-65.319,-176.797,6.945,148.353
C03063=1207.684,275.547,-65.348,-176.794,6.948,148.353
C03064=1207.680,275.796,-65.376,-176.792,6.949,148.353
C03065=1207.676,276.044,-65.404,-176.789,6.952,148.353
C03066=1207.671,276.293,-65.432,-176.787,6.955,148.353
C03067=1207.667,276.541,-65.460,-176.784,6.957,148.352
C03068=1207.662,276.790,-65.489,-176.782,6.960,148.352
C03069=1207.658,277.037,-65.517,-176.779,6.963,148.352
C03070=1207.653,277.286,-65.546,-176.777,6.965,148.352
C03071=1207.649,277.534,-65.573,-176.774,6.967,148.352
C03072=1207.645,277.783,-65.601,-176.772,6.970,148.352
C03073=1207.640,278.031,-65.630,-176.769,6.972,148.352
C03074=1207.636,278.280,-65.658,-176.766,6.975,148.352
C03075=1207.632,278.528,-65.687,-176.764,6.977,148.351
C03076=1207.628,278.776,-65.714,-176.761,6.980,148.351
C03077=1207.623,279.025,-65.743,-176.759,6.982,148.351
C03078=1207.619,279.273,-65.771,-176.757,6.984,148.351
C03079=1207.614,279.522,-65.800,-176.754,6.987,148.351
C03080=1207.610,279.770,-65.828,-176.751,6.989,148.351
C03081=1207.605,280.019,-65.856,-176.749,6.992,148.351
C03082=1207.601,280.266,-65.885,-176.747,6.994,148.351
C03083=1207.597,280.515,-65.913,-176.744,6.997,148.351
C03084=1207.593,280.763,-65.942,-176.741,6.999,148.350
C03085=1207.588,281.012,-65.970,-176.739,7.001,148.350
C03086=1207.584,281.260,-65.999,-176.736,7.004,148.350
C03087=1207.579,281.508,-66.027,-176.734,7.006,148.350
C03088=1207.575,281.757,-66.056,-176.731,7.009,148.350
C03089=1207.571,282.005,-66.084,-176.729,7.011,148.350
C03090=1207.566,282.253,-66.112,-176.726,7.014,148.350
C03091=1207.563,282.501,-66.141,-176.724,7.016,148.350
C03092=1207.558,282.750,-66.170,-176.721,7.019,148.350
C03093=1207.553,282.998,-66.198,-176.719,7.021,148.349
C03094=1207.549,283.247,-66.227,-176.717,7.023,148.349
C03095=1207.545,283.495,-66.256,-176.714,7.026,148.349
C03096=1207.540,283.743,-66.284,-176.711,7.028,148.349
C03097=1207.536,283.991,-66.312,-176.709,7.031,148.349
C03098=1207.532,284.240,-66.342,-176.707,7.034,148.349
C03099=1207.527,284.488,-66.370,-176.703,7.036,148.349
C03100=1207.523,284.736,-66.398,-176.701,7.038,148.349
C03101=1207.519,284.985,-66.428,-176.699,7.041,148.349
C03102=1207.514,285.234,-66.456,-176.696,7.044,148.349
C03103=1207.510,285.481,-66.485,-176.694,7.047,148.349
C03104=1207.506,285.730,-66.514,-176.691,7.049,148.348
C03105=1207.501,285.979,-66.542,-176.688,7.052,148.348
C03106=1207.496,286.226,-66.571,-176.686,7.054,148.348
C03107=1207.493,286.475,-66.600,-176.684,7.057,148.348
C03108=1207.488,286.723,-66.629,-176.681,7.059,148.348
C03109=1207.483,286.971,-66.657,-176.678,7.062,148.348
C03110=1207.480,287.219,-66.686,-176.676,7.064,148.348
C03111=1207.475,287.468,-66.715,-176.674,7.066,148.348
C03112=1207.471,287.716,-66.744,-176.671,7.069,148.348
C03113=1207.466,287.964,-66.773,-176.669,7.071,148.347
C03114=1207.462,288.213,-66.802,-176.666,7.074,148.347
C03115=1207.458,288.461,-66.830,-176.664,7.076,148.347
C03116=1207.454,288.735,-66.863,-176.661,7.079,148.347
C03117=1207.448,289.010,-66.895,-176.658,7.082,148.347
C03118=1207.443,289.284,-66.927,-176.655,7.085,148.347
C03119=1207.439,289.558,-66.959,-176.653,7.088,148.347
C03120=1207.434,289.807,-66.988,-176.651,7.090,148.347
C03121=1207.430,290.055,-67.017,-176.648,7.093,148.347
C03122=1207.425,290.303,-67.046,-176.645,7.095,148.347
C03123=1207.422,290.551,-67.074,-176.643,7.098,148.347
C03124=1207.417,290.799,-67.104,-176.640,7.100,148.346
C03125=1207.413,291.048,-67.133,-176.638,7.103,148.346
C03126=1207.408,291.296,-67.162,-176.636,7.105,148.346
C03127=1207.404,291.544,-67.191,-176.633,7.109,148.346
C03128=1207.400,291.792,-67.221,-176.630,7.110,148.346
C03129=1207.395,292.041,-67.249,-176.628,7.113,148.346
C03130=1207.391,292.290,-67.279,-176.626,7.116,148.346
C03131=1207.387,292.537,-67.307,-176.623,7.119,148.346
C03132=1207.383,292.785,-67.337,-176.621,7.121,148.346
C03133=1207.378,293.034,-67.365,-176.618,7.124,148.346
C03134=1207.374,293.282,-67.395,-176.616,7.126,148.346
C03135=1207.370,293.530,-67.424,-176.613,7.129,148.346
C03136=1207.366,293.779,-67.454,-176.611,7.131,148.346
C03137=1207.361,294.026,-67.483,-176.608,7.134,148.346
C03138=1207.357,294.275,-67.512,-176.606,7.136,148.345
C03139=1207.352,294.523,-67.541,-176.603,7.139,148.345
C03140=1207.348,294.772,-67.571,-176.600,7.142,148.345
C03141=1207.344,295.020,-67.600,-176.598,7.144,148.345
C03142=1207.340,295.268,-67.629,-176.596,7.147,148.345
C03143=1207.335,295.516,-67.659,-176.594,7.150,148.345
C03144=1207.331,295.764,-67.688,-176.591,7.153,148.345
C03145=1207.327,296.012,-67.717,-176.588,7.155,148.345
C03146=1207.323,296.261,-67.747,-176.586,7.158,148.345
C03147=1207.318,296.509,-67.776,-176.583,7.160,148.345
C03148=1207.314,296.758,-67.805,-176.581,7.163,148.345
C03149=1207.310,297.006,-67.835,-176.579,7.165,148.345
C03150=1207.305,297.254,-67.864,-176.576,7.168,148.345
C03151=1207.301,297.503,-67.893,-176.574,7.170,148.345
C03152=1207.297,297.750,-67.923,-176.571,7.173,148.345
C03153=1207.292,297.999,-67.953,-176.569,7.175,148.345
C03154=1207.287,298.247,-67.982,-176.566,7.178,148.345
C03155=1207.284,298.495,-68.012,-176.564,7.181,148.345
C03156=1207.279,298.743,-68.042,-176.561,7.184,148.345
C03157=1207.275,298.991,-68.071,-176.559,7.187,148.345
C03158=1207.271,299.239,-68.101,-176.557,7.189,148.344
C03159=1207.267,299.488,-68.130,-176.554,7.192,148.344
C03160=1207.263,299.736,-68.159,-176.552,7.194,148.344
C03161=1207.258,299.985,-68.190,-176.549,7.197,148.344
C03162=1207.254,300.233,-68.219,-176.547,7.199,148.344
C03163=1207.249,300.481,-68.248,-176.544,7.202,148.344
C03164=1207.245,300.729,-68.278,-176.542,7.204,148.344
C03165=1207.241,300.977,-68.308,-176.539,7.207,148.344
C03166=1207.236,301.226,-68.338,-176.537,7.210,148.344
C03167=1207.232,301.474,-68.368,-176.534,7.213,148.344
C03168=1207.228,301.722,-68.397,-176.532,7.216,148.344
C03169=1207.223,301.970,-68.426,-176.529,7.218,148.344
C03170=1207.219,302.217,-68.456,-176.527,7.221,148.344
C03171=1207.214,302.466,-68.486,-176.525,7.223,148.344
C03172=1207.210,302.714,-68.516,-176.522,7.226,148.344
C03173=1207.206,302.962,-68.545,-176.520,7.228,148.344
C03174=1207.202,303.210,-68.575,-176.517,7.231,148.344
C03175=1207.197,303.459,-68.605,-176.514,7.234,148.344
C03176=1207.193,303.707,-68.635,-176.512,7.236,148.344
C03177=1207.189,303.955,-68.664,-176.510,7.240,148.344
C03178=1207.184,304.203,-68.695,-176.508,7.242,148.344
C03179=1207.181,304.452,-68.725,-176.505,7.245,148.344
C03180=1207.177,304.700,-68.754,-176.503,7.247,148.344
C03181=1207.173,304.948,-68.785,-176.500,7.250,148.344
C03182=1207.168,305.197,-68.815,-176.498,7.252,148.344
C03183=1207.164,305.444,-68.845,-176.496,7.255,148.344
C03184=1207.160,305.693,-68.874,-176.493,7.259,148.344
C03185=1207.155,305.941,-68.904,-176.491,7.261,148.344
C03186=1207.151,306.189,-68.934,-176.488,7.264,148.344
C03187=1207.146,306.437,-68.964,-176.486,7.266,148.343
C03188=1207.142,306.685,-68.995,-176.483,7.269,148.343
C03189=1207.138,306.933,-69.024,-176.481,7.271,148.343
C03190=1207.133,307.181,-69.055,-176.479,7.274,148.343
C03191=1207.129,307.429,-69.084,-176.476,7.277,148.343
C03192=1207.125,307.677,-69.114,-176.474,7.279,148.343
C03193=1207.120,307.926,-69.145,-176.471,7.282,148.343
C03194=1207.116,308.173,-69.175,-176.469,7.285,148.344
C03195=1207.112,308.423,-69.205,-176.467,7.288,148.343
C03196=1207.108,308.670,-69.235,-176.464,7.291,148.343
C03197=1207.103,308.919,-69.265,-176.462,7.293,148.343
C03198=1207.099,309.166,-69.296,-176.459,7.296,148.343
C03199=1207.095,309.415,-69.326,-176.457,7.298,148.343
C03200=1207.091,309.663,-69.356,-176.454,7.301,148.343
C03201=1207.087,309.910,-69.386,-176.452,7.304,148.343
C03202=1207.082,310.159,-69.416,-176.450,7.307,148.344
C03203=1207.079,310.407,-69.446,-176.447,7.310,148.343
C03204=1207.074,310.656,-69.477,-176.445,7.312,148.343
C03205=1207.070,310.904,-69.507,-176.443,7.315,148.343
C03206=1207.065,311.151,-69.537,-176.440,7.317,148.343
C03207=1207.061,311.400,-69.567,-176.438,7.321,148.343
C03208=1207.056,311.648,-69.598,-176.435,7.324,148.343
C03209=1207.052,311.896,-69.628,-176.433,7.326,148.344
C03210=1207.048,312.145,-69.658,-176.431,7.329,148.344
C03211=1207.044,312.393,-69.689,-176.429,7.331,148.343
C03212=1207.040,312.640,-69.719,-176.426,7.334,148.343
C03213=1207.035,312.888,-69.750,-176.423,7.337,148.343
C03214=1207.031,313.136,-69.779,-176.421,7.340,148.343
C03215=1207.027,313.385,-69.811,-176.419,7.343,148.344
C03216=1207.023,313.633,-69.841,-176.417,7.345,148.344
C03217=1207.018,313.881,-69.871,-176.414,7.348,148.344
C03218=1207.014,314.129,-69.902,-176.411,7.351,148.344
C03219=1207.010,314.377,-69.932,-176.409,7.353,148.343
C03220=1207.005,314.653,-69.966,-176.407,7.357,148.344
C03221=1207.001,314.929,-70.001,-176.404,7.360,148.344
C03222=1206.996,315.206,-70.034,-176.402,7.363,148.344
C03223=1206.991,315.481,-70.068,-176.399,7.366,148.344
C03224=1206.987,315.729,-70.099,-176.396,7.369,148.344
C03225=1206.983,315.978,-70.130,-176.394,7.371,148.344
C03226=1206.978,316.226,-70.160,-176.392,7.374,148.344
C03227=1206.974,316.474,-70.190,-176.389,7.377,148.344
C03228=1206.970,316.722,-70.221,-176.387,7.380,148.344
C03229=1206.965,316.971,-70.252,-176.385,7.383,148.344
C03230=1206.961,317.219,-70.283,-176.383,7.385,148.344
C03231=1206.957,317.466,-70.313,-176.380,7.388,148.344
C03232=1206.952,317.714,-70.344,-176.378,7.391,148.344
C03233=1206.948,317.963,-70.375,-176.375,7.393,148.344
C03234=1206.945,318.210,-70.405,-176.373,7.397,148.344
C03235=1206.940,318.458,-70.436,-176.371,7.399,148.344
C03236=1206.936,318.707,-70.467,-176.368,7.402,148.344
C03237=1206.931,318.955,-70.498,-176.366,7.405,148.344
C03238=1206.927,319.203,-70.528,-176.364,7.408,148.344
C03239=1206.923,319.451,-70.559,-176.361,7.411,148.344
C03240=1206.919,319.699,-70.590,-176.360,7.413,148.344
C03241=1206.914,319.947,-70.621,-176.357,7.416,148.344
C03242=1206.910,320.195,-70.652,-176.354,7.419,148.344
C03243=1206.907,320.443,-70.682,-176.353,7.422,148.345
C03244=1206.902,320.691,-70.713,-176.350,7.425,148.345
C03245=1206.898,320.940,-70.744,-176.347,7.428,148.345
C03246=1206.893,321.188,-70.775,-176.346,7.430,148.345
C03247=1206.889,321.435,-70.806,-176.343,7.433,148.345
C03248=1206.886,321.683,-70.837,-176.341,7.435,148.345
C03249=1206.881,321.931,-70.868,-176.339,7.439,148.345
C03250=1206.877,322.179,-70.899,-176.336,7.442,148.345
C03251=1206.873,322.428,-70.930,-176.334,7.444,148.345
C03252=1206.868,322.675,-70.961,-176.332,7.447,148.345
C03253=1206.864,322.923,-70.992,-176.330,7.450,148.345
C03254=1206.860,323.172,-71.023,-176.327,7.453,148.345
C03255=1206.856,323.419,-71.053,-176.325,7.456,148.345
C03256=1206.852,323.667,-71.085,-176.323,7.458,148.345
C03257=1206.847,323.915,-71.116,-176.320,7.462,148.345
C03258=1206.843,324.163,-71.147,-176.318,7.465,148.345
C03259=1206.839,324.412,-71.178,-176.315,7.467,148.345
C03260=1206.834,324.659,-71.209,-176.313,7.470,148.346
C03261=1206.830,324.908,-71.240,-176.311,7.472,148.345
C03262=1206.826,325.156,-71.271,-176.309,7.476,148.346
C03263=1206.822,325.404,-71.303,-176.306,7.479,148.346
C03264=1206.818,325.652,-71.334,-176.305,7.481,148.346
C03265=1206.813,325.899,-71.365,-176.302,7.484,148.346
C03266=1206.809,326.148,-71.396,-176.300,7.486,148.346
C03267=1206.805,326.396,-71.427,-176.298,7.490,148.346
C03268=1206.801,326.644,-71.459,-176.295,7.493,148.346
C03269=1206.796,326.892,-71.490,-176.293,7.495,148.346
C03270=1206.793,327.140,-71.522,-176.291,7.498,148.346
C03271=1206.788,327.388,-71.552,-176.288,7.502,148.346
C03272=1206.784,327.636,-71.584,-176.286,7.504,148.346
C03273=1206.780,327.884,-71.615,-176.284,7.507,148.347
C03274=1206.776,328.132,-71.647,-176.282,7.509,148.347
C03275=1206.771,328.380,-71.678,-176.280,7.513,148.347
C03276=1206.768,328.628,-71.709,-176.277,7.516,148.347
C03277=1206.763,328.876,-71.740,-176.275,7.518,148.347
C03278=1206.759,329.123,-71.772,-176.273,7.521,148.347
C03279=1206.755,329.372,-71.803,-176.270,7.525,148.347
C03280=1206.750,329.619,-71.834,-176.268,7.527,148.347
C03281=1206.746,329.868,-71.865,-176.266,7.530,148.347
C03282=1206.742,330.115,-71.897,-176.264,7.532,148.347
C03283=1206.738,330.363,-71.929,-176.262,7.536,148.348
C03284=1206.734,330.612,-71.960,-176.260,7.539,148.348
C03285=1206.729,330.860,-71.992,-176.257,7.541,148.348
C03286=1206.725,331.108,-72.023,-176.255,7.545,148.348
C03287=1206.721,331.356,-72.054,-176.253,7.547,148.348
C03288=1206.717,331.604,-72.086,-176.251,7.550,148.348
C03289=1206.713,331.852,-72.117,-176.248,7.553,148.348
C03290=1206.709,332.100,-72.149,-176.247,7.556,148.348
C03291=1206.704,332.347,-72.181,-176.244,7.559,148.348
C03292=1206.700,332.595,-72.213,-176.242,7.562,148.348
C03293=1206.696,332.843,-72.244,-176.240,7.565,148.349
C03294=1206.692,333.091,-72.275,-176.237,7.568,148.349
C03295=1206.688,333.339,-72.307,-176.236,7.570,148.349
C03296=1206.683,333.588,-72.339,-176.233,7.574,148.349
C03297=1206.679,333.836,-72.371,-176.231,7.577,148.349
C03298=1206.675,334.083,-72.402,-176.229,7.579,148.349
C03299=1206.671,334.331,-72.434,-176.227,7.582,148.349
C03300=1206.666,334.579,-72.466,-176.224,7.586,148.349
C03301=1206.662,334.827,-72.497,-176.223,7.588,148.350
C03302=1206.658,335.075,-72.529,-176.220,7.591,148.350
C03303=1206.654,335.323,-72.560,-176.218,7.594,148.350
C03304=1206.650,335.571,-72.593,-176.216,7.597,148.350
C03305=1206.645,335.818,-72.624,-176.214,7.600,148.350
C03306=1206.642,336.066,-72.656,-176.212,7.602,148.350
C03307=1206.638,336.314,-72.688,-176.210,7.606,148.350
C03308=1206.632,336.563,-72.719,-176.208,7.608,148.351
C03309=1206.629,336.811,-72.751,-176.205,7.611,148.351
C03310=1206.625,337.059,-72.783,-176.203,7.615,148.351
C03311=1206.620,337.306,-72.815,-176.201,7.617,148.351
C03312=1206.616,337.554,-72.847,-176.199,7.621,148.351
C03313=1206.613,337.803,-72.879,-176.196,7.624,148.351
C03314=1206.608,338.050,-72.911,-176.195,7.626,148.351
C03315=1206.604,338.298,-72.943,-176.193,7.629,148.352
C03316=1206.600,338.546,-72.975,-176.191,7.632,148.352
C03317=1206.595,338.794,-73.007,-176.188,7.635,148.352
C03318=1206.591,339.042,-73.038,-176.186,7.638,148.352
C03319=1206.588,339.290,-73.070,-176.184,7.641,148.352
C03320=1206.583,339.538,-73.102,-176.182,7.644,148.352
C03321=1206.579,339.786,-73.134,-176.180,7.647,148.353
C03322=1206.575,340.034,-73.167,-176.178,7.650,148.353
C03323=1206.570,340.281,-73.198,-176.176,7.653,148.353
C03324=1206.566,340.560,-73.235,-176.173,7.656,148.353
C03325=1206.561,340.837,-73.270,-176.171,7.660,148.353
C03326=1206.557,341.116,-73.307,-176.169,7.663,148.354
C03327=1206.552,341.394,-73.342,-176.166,7.666,148.354
C03328=1206.548,341.642,-73.374,-176.165,7.669,148.354
C03329=1206.543,341.890,-73.407,-176.162,7.672,148.354
C03330=1206.539,342.138,-73.439,-176.160,7.675,148.354
C03331=1206.535,342.386,-73.471,-176.159,7.678,148.354
C03332=1206.531,342.634,-73.503,-176.156,7.681,148.355
C03333=1206.526,342.882,-73.535,-176.155,7.684,148.355
C03334=1206.523,343.129,-73.568,-176.152,7.687,148.355
C03335=1206.518,343.377,-73.600,-176.150,7.690,148.355
C03336=1206.515,343.625,-73.632,-176.148,7.693,148.355
C03337=1206.510,343.873,-73.664,-176.146,7.696,148.355
C03338=1206.506,344.120,-73.697,-176.144,7.698,148.356
C03339=1206.502,344.369,-73.729,-176.142,7.702,148.356
C03340=1206.498,344.617,-73.761,-176.140,7.705,148.356
C03341=1206.493,344.864,-73.793,-176.138,7.708,148.356
C03342=1206.489,345.112,-73.826,-176.136,7.711,148.356
C03343=1206.485,345.360,-73.858,-176.134,7.713,148.357
C03344=1206.481,345.609,-73.891,-176.132,7.717,148.357
C03345=1206.477,345.855,-73.923,-176.130,7.720,148.357
C03346=1206.472,346.104,-73.955,-176.128,7.723,148.357
C03347=1206.468,346.352,-73.988,-176.126,7.726,148.357
C03348=1206.464,346.599,-74.020,-176.124,7.729,148.358
C03349=1206.460,346.848,-74.053,-176.122,7.732,148.358
C03350=1206.456,347.095,-74.084,-176.120,7.735,148.358
C03351=1206.452,347.343,-74.117,-176.118,7.738,148.358
C03352=1206.447,347.591,-74.150,-176.116,7.741,148.358
C03353=1206.444,347.839,-74.182,-176.114,7.744,148.359
C03354=1206.439,348.087,-74.215,-176.112,7.747,148.359
C03355=1206.435,348.335,-74.248,-176.110,7.750,148.359
C03356=1206.431,348.582,-74.279,-176.108,7.753,148.359
C03357=1206.427,348.830,-74.312,-176.106,7.756,148.359
C03358=1206.422,349.078,-74.345,-176.104,7.759,148.360
C03359=1206.419,349.326,-74.377,-176.102,7.762,148.360
C03360=1206.414,349.574,-74.410,-176.101,7.765,148.360
C03361=1206.410,349.822,-74.443,-176.098,7.768,148.360
C03362=1206.407,350.070,-74.475,-176.097,7.771,148.361
C03363=1206.402,350.317,-74.508,-176.095,7.774,148.361
C03364=1206.397,350.565,-74.540,-176.093,7.777,148.361
C03365=1206.393,350.813,-74.573,-176.091,7.780,148.361
C03366=1206.390,351.061,-74.605,-176.089,7.783,148.362
C03367=1206.385,351.309,-74.638,-176.087,7.786,148.362
C03368=1206.381,351.556,-74.671,-176.085,7.789,148.362
C03369=1206.377,351.805,-74.704,-176.083,7.793,148.362
C03370=1206.373,352.052,-74.736,-176.082,7.795,148.363
C03371=1206.369,352.300,-74.769,-176.079,7.799,148.363
C03372=1206.364,352.547,-74.802,-176.078,7.801,148.363
C03373=1206.360,352.795,-74.835,-176.075,7.804,148.363
C03374=1206.356,353.043,-74.867,-176.074,7.807,148.364
C03375=1206.352,353.291,-74.900,-176.072,7.811,148.364
C03376=1206.348,353.539,-74.933,-176.070,7.814,148.364
C03377=1206.344,353.787,-74.965,-176.068,7.816,148.364
C03378=1206.340,354.035,-74.999,-176.066,7.820,148.365
C03379=1206.336,354.282,-75.031,-176.065,7.823,148.365
C03380=1206.332,354.530,-75.064,-176.063,7.826,148.365
C03381=1206.328,354.778,-75.097,-176.061,7.828,148.365
C03382=1206.323,355.026,-75.130,-176.059,7.832,148.366
C03383=1206.319,355.274,-75.163,-176.057,7.835,148.366
C03384=1206.315,355.521,-75.196,-176.055,7.838,148.366
C03385=1206.311,355.770,-75.229,-176.053,7.842,148.367
C03386=1206.307,356.017,-75.261,-176.052,7.844,148.367
C03387=1206.303,356.265,-75.294,-176.050,7.847,148.367
C03388=1206.299,356.513,-75.328,-176.048,7.850,148.367
C03389=1206.295,356.760,-75.361,-176.046,7.854,148.368
C03390=1206.291,357.008,-75.394,-176.045,7.856,148.368
C03391=1206.286,357.256,-75.426,-176.043,7.860,148.368
C03392=1206.282,357.504,-75.459,-176.041,7.862,148.368
C03393=1206.278,357.752,-75.493,-176.039,7.866,148.369
C03394=1206.274,358.000,-75.526,-176.038,7.868,148.369
C03395=1206.270,358.247,-75.559,-176.035,7.872,148.369
C03396=1206.266,358.495,-75.592,-176.034,7.875,148.370
C03397=1206.262,358.743,-75.625,-176.032,7.878,148.370
C03398=1206.258,358.990,-75.658,-176.030,7.881,148.370
C03399=1206.254,359.238,-75.691,-176.029,7.884,148.370
C03400=1206.250,359.486,-75.724,-176.026,7.887,148.371
C03401=1206.246,359.733,-75.757,-176.025,7.890,148.371
C03402=1206.242,359.981,-75.790,-176.023,7.894,148.371
C03403=1206.237,360.229,-75.824,-176.022,7.896,148.372
C03404=1206.233,360.477,-75.857,-176.020,7.900,148.372
C03405=1206.229,360.724,-75.890,-176.018,7.903,148.372
C03406=1206.225,360.972,-75.923,-176.016,7.906,148.373
C03407=1206.221,361.220,-75.956,-176.015,7.909,148.373
C03408=1206.217,361.468,-75.989,-176.013,7.912,148.373
C03409=1206.213,361.715,-76.022,-176.012,7.915,148.374
C03410=1206.208,361.963,-76.056,-176.010,7.918,148.374
C03411=1206.204,362.211,-76.089,-176.008,7.921,148.374
C03412=1206.200,362.458,-76.122,-176.007,7.924,148.375
C03413=1206.196,362.706,-76.155,-176.005,7.927,148.375
C03414=1206.192,362.955,-76.189,-176.004,7.930,148.375
C03415=1206.188,363.203,-76.222,-176.002,7.934,148.376
C03416=1206.184,363.450,-76.256,-176.000,7.936,148.376
C03417=1206.180,363.697,-76.289,-175.998,7.940,148.376
C03418=1206.176,363.945,-76.323,-175.997,7.942,148.376
C03419=1206.171,364.193,-76.356,-175.995,7.946,148.377
C03420=1206.167,364.441,-76.389,-175.994,7.949,148.377
C03421=1206.163,364.688,-76.422,-175.992,7.951,148.377
C03422=1206.159,364.936,-76.456,-175.990,7.955,148.378
C03423=1206.156,365.184,-76.489,-175.989,7.958,148.378
C03424=1206.152,365.432,-76.523,-175.987,7.961,148.379
C03425=1206.147,365.680,-76.556,-175.986,7.964,148.379
C03426=1206.143,365.927,-76.590,-175.984,7.967,148.379
C03427=1206.139,366.175,-76.623,-175.983,7.970,148.380
C03428=1206.135,366.455,-76.661,-175.981,7.974,148.380
C03429=1206.130,366.736,-76.699,-175.980,7.977,148.381
C03430=1206.125,367.016,-76.737,-175.978,7.980,148.381
C03431=1206.120,367.296,-76.775,-175.976,7.984,148.381
C03432=1206.116,367.544,-76.808,-175.975,7.987,148.382
C03433=1206.112,367.792,-76.841,-175.973,7.990,148.382
C03434=1206.108,368.040,-76.876,-175.972,7.993,148.382
C03435=1206.104,368.288,-76.909,-175.970,7.997,148.383
C03436=1206.100,368.535,-76.943,-175.969,7.999,148.383
C03437=1206.096,368.782,-76.976,-175.967,8.002,148.383
C03438=1206.092,369.030,-77.010,-175.966,8.005,148.384
C03439=1206.087,369.278,-77.043,-175.964,8.008,148.384
C03440=1206.084,369.526,-77.078,-175.963,8.011,148.385
C03441=1206.080,369.774,-77.111,-175.962,8.014,148.385
C03442=1206.076,370.021,-77.145,-175.960,8.018,148.386
C03443=1206.071,370.269,-77.178,-175.959,8.020,148.386
C03444=1206.067,370.517,-77.211,-175.957,8.023,148.386
C03445=1206.064,370.764,-77.246,-175.956,8.027,148.387
C03446=1206.059,371.012,-77.279,-175.954,8.030,148.387
C03447=1206.055,371.260,-77.313,-175.953,8.033,148.388
C03448=1206.051,371.507,-77.346,-175.952,8.035,148.388
C03449=1206.047,371.754,-77.380,-175.950,8.039,148.388
C03450=1206.043,372.003,-77.414,-175.949,8.042,148.389
C03451=1206.039,372.250,-77.448,-175.948,8.045,148.389
C03452=1206.035,372.498,-77.482,-175.947,8.047,148.390
C03453=1206.030,372.745,-77.516,-175.945,8.051,148.390
C03454=1206.027,372.994,-77.549,-175.944,8.054,148.390
C03455=1206.023,373.241,-77.583,-175.942,8.057,148.391
C03456=1206.018,373.489,-77.617,-175.941,8.060,148.391
C03457=1206.014,373.736,-77.651,-175.940,8.062,148.392
C03458=1206.010,373.985,-77.685,-175.938,8.066,148.392
C03459=1206.006,374.232,-77.719,-175.938,8.069,148.393
C03460=1206.002,374.479,-77.753,-175.936,8.072,148.393
C03461=1205.998,374.727,-77.786,-175.935,8.075,148.393
C03462=1205.994,374.975,-77.821,-175.934,8.078,148.394
C03463=1205.990,375.223,-77.854,-175.933,8.080,148.394
C03464=1205.986,375.470,-77.888,-175.931,8.084,148.395
C03465=1205.981,375.717,-77.922,-175.930,8.087,148.395
C03466=1205.978,375.966,-77.956,-175.929,8.090,148.396
C03467=1205.973,376.213,-77.990,-175.928,8.093,148.396
C03468=1205.969,376.460,-78.024,-175.927,8.095,148.396
C03469=1205.966,376.709,-78.058,-175.925,8.098,148.397
C03470=1205.961,376.956,-78.092,-175.924,8.101,148.397
C03471=1205.958,377.203,-78.126,-175.923,8.104,148.398
C03472=1205.953,377.451,-78.160,-175.922,8.107,148.398
C03473=1205.949,377.699,-78.194,-175.921,8.110,148.398
C03474=1205.945,377.946,-78.228,-175.919,8.113,148.399
C03475=1205.941,378.194,-78.262,-175.918,8.117,148.400
C03476=1205.937,378.442,-78.296,-175.917,8.119,148.400
C03477=1205.933,378.689,-78.330,-175.916,8.122,148.400
C03478=1205.929,378.936,-78.364,-175.915,8.125,148.401
C03479=1205.925,379.185,-78.398,-175.914,8.128,148.401
C03480=1205.921,379.432,-78.432,-175.913,8.131,148.402
C03481=1205.916,379.680,-78.467,-175.912,8.134,148.402
C03482=1205.913,379.927,-78.501,-175.911,8.137,148.403
C03483=1205.908,380.176,-78.535,-175.910,8.140,148.403
C03484=1205.904,380.423,-78.569,-175.909,8.143,148.404
C03485=1205.900,380.671,-78.603,-175.908,8.146,148.404
C03486=1205.897,380.918,-78.637,-175.907,8.149,148.405
C03487=1205.892,381.165,-78.672,-175.906,8.151,148.405
C03488=1205.889,381.414,-78.705,-175.904,8.154,148.405
C03489=1205.884,381.661,-78.740,-175.904,8.157,148.406
C03490=1205.880,381.908,-78.774,-175.903,8.159,148.406
C03491=1205.876,382.156,-78.808,-175.902,8.162,148.407
C03492=1205.872,382.403,-78.842,-175.901,8.165,148.407
C03493=1205.868,382.651,-78.877,-175.900,8.168,148.408
C03494=1205.863,382.900,-78.911,-175.899,8.171,148.408
C03495=1205.860,383.147,-78.945,-175.898,8.174,148.409
C03496=1205.855,383.394,-78.979,-175.897,8.177,148.409
C03497=1205.852,383.642,-79.013,-175.896,8.180,148.410
C03498=1205.847,383.889,-79.048,-175.895,8.183,148.410
C03499=1205.844,384.137,-79.082,-175.894,8.185,148.411
C03500=1205.839,384.385,-79.117,-175.894,8.188,148.411
C03501=1205.836,384.632,-79.150,-175.893,8.191,148.412
C03502=1205.832,384.880,-79.185,-175.892,8.194,148.412
C03503=1205.827,385.127,-79.220,-175.891,8.197,148.413
C03504=1205.824,385.375,-79.254,-175.890,8.200,148.413
C03505=1205.819,385.623,-79.288,-175.890,8.202,148.414
C03506=1205.815,385.870,-79.322,-175.888,8.205,148.414
C03507=1205.812,386.118,-79.357,-175.888,8.208,148.415
C03508=1205.807,386.365,-79.392,-175.886,8.211,148.415
C03509=1205.804,386.613,-79.426,-175.886,8.214,148.416
C03510=1205.799,386.860,-79.460,-175.885,8.216,148.416
C03511=1205.795,387.108,-79.495,-175.884,8.219,148.417
C03512=1205.791,387.356,-79.529,-175.883,8.222,148.417
C03513=1205.787,387.603,-79.564,-175.883,8.224,148.418
C03514=1205.784,387.851,-79.598,-175.882,8.227,148.418
C03515=1205.779,388.098,-79.632,-175.881,8.230,148.419
C03516=1205.774,388.346,-79.667,-175.880,8.233,148.419
C03517=1205.771,388.593,-79.701,-175.880,8.235,148.420
C03518=1205.767,388.841,-79.735,-175.879,8.238,148.420
C03519=1205.763,389.089,-79.770,-175.878,8.241,148.421
C03520=1205.759,389.336,-79.804,-175.878,8.244,148.421
C03521=1205.755,389.584,-79.839,-175.876,8.246,148.422
C03522=1205.750,389.832,-79.873,-175.876,8.250,148.422
C03523=1205.747,390.079,-79.908,-175.875,8.252,148.422
C03524=1205.742,390.327,-79.942,-175.874,8.255,148.423
C03525=1205.738,390.574,-79.977,-175.873,8.258,148.424
C03526=1205.734,390.822,-80.012,-175.873,8.260,148.424
C03527=1205.730,391.069,-80.046,-175.872,8.263,148.425
C03528=1205.726,391.317,-80.081,-175.872,8.265,148.425
C03529=1205.722,391.564,-80.115,-175.871,8.268,148.426
C03530=1205.719,391.812,-80.150,-175.870,8.270,148.426
C03531=1205.714,392.060,-80.184,-175.870,8.273,148.427
C03532=1205.710,392.342,-80.224,-175.869,8.276,148.427
C03533=1205.705,392.625,-80.263,-175.868,8.280,148.428
C03534=1205.701,392.907,-80.303,-175.867,8.283,148.428
C03535=1205.696,393.190,-80.342,-175.867,8.286,148.429
C03536=1205.692,393.437,-80.377,-175.866,8.288,148.429
C03537=1205.688,393.685,-80.412,-175.865,8.291,148.430
C03538=1205.684,393.933,-80.446,-175.865,8.293,148.430
C03539=1205.680,394.181,-80.481,-175.864,8.296,148.431
C03540=1205.676,394.427,-80.516,-175.863,8.298,148.431
C03541=1205.672,394.675,-80.551,-175.863,8.301,148.432
C03542=1205.667,394.923,-80.585,-175.863,8.304,148.433
C03543=1205.664,395.171,-80.620,-175.862,8.307,148.433
C03544=1205.660,395.418,-80.654,-175.861,8.309,148.433
C03545=1205.656,395.666,-80.689,-175.861,8.311,148.434
C03546=1205.651,395.913,-80.724,-175.860,8.314,148.435
C03547=1205.647,396.161,-80.759,-175.860,8.316,148.435
C03548=1205.644,396.408,-80.792,-175.859,8.319,148.436
C03549=1205.640,396.656,-80.828,-175.858,8.321,148.436
C03550=1205.635,396.903,-80.862,-175.858,8.324,148.437
C03551=1205.631,397.151,-80.897,-175.857,8.327,148.437
C03552=1205.627,397.398,-80.932,-175.857,8.329,148.438
C03553=1205.623,397.646,-80.967,-175.856,8.332,148.438
C03554=1205.619,397.893,-81.001,-175.856,8.334,148.439
C03555=1205.616,398.141,-81.037,-175.856,8.336,148.439
C03556=1205.611,398.388,-81.071,-175.855,8.339,148.440
C03557=1205.607,398.636,-81.106,-175.854,8.341,148.440
C03558=1205.603,398.883,-81.141,-175.854,8.344,148.441
C03559=1205.599,399.131,-81.176,-175.853,8.347,148.441
C03560=1205.595,399.378,-81.210,-175.853,8.349,148.442
C03561=1205.591,399.626,-81.245,-175.852,8.351,148.442
C03562=1205.587,399.873,-81.280,-175.852,8.354,148.443
C03563=1205.583,400.121,-81.315,-175.851,8.356,148.443
C03564=1205.579,400.369,-81.350,-175.851,8.359,148.444
C03565=1205.575,400.616,-81.385,-175.850,8.362,148.444
C03566=1205.571,400.864,-81.419,-175.850,8.364,148.445
C03567=1205.567,401.111,-81.454,-175.849,8.366,148.445
C03568=1205.563,401.359,-81.489,-175.849,8.368,148.446
C03569=1205.559,401.606,-81.524,-175.848,8.371,148.446
C03570=1205.555,401.854,-81.559,-175.848,8.373,148.447
C03571=1205.550,402.101,-81.594,-175.848,8.376,148.447
C03572=1205.547,402.349,-81.629,-175.847,8.378,148.448
C03573=1205.543,402.597,-81.664,-175.847,8.381,148.448
C03574=1205.539,402.844,-81.699,-175.846,8.383,148.449
C03575=1205.535,403.092,-81.733,-175.846,8.385,148.449
C03576=1205.531,403.338,-81.768,-175.846,8.387,148.450
C03577=1205.527,403.587,-81.803,-175.845,8.390,148.450
C03578=1205.522,403.834,-81.838,-175.845,8.393,148.451
C03579=1205.519,404.081,-81.873,-175.844,8.395,148.451
C03580=1205.515,404.330,-81.908,-175.844,8.397,148.452
C03581=1205.511,404.576,-81.943,-175.843,8.399,148.452
C03582=1205.507,404.825,-81.978,-175.843,8.402,148.453
C03583=1205.502,405.071,-82.013,-175.843,8.404,148.453
C03584=1205.498,405.319,-82.048,-175.842,8.407,148.454
C03585=1205.494,405.566,-82.083,-175.842,8.409,148.454
C03586=1205.490,405.814,-82.118,-175.841,8.411,148.455
C03587=1205.487,406.062,-82.153,-175.841,8.414,148.455
C03588=1205.483,406.309,-82.188,-175.841,8.416,148.456
C03589=1205.479,406.556,-82.223,-175.840,8.418,148.456
C03590=1205.474,406.804,-82.258,-175.840,8.420,148.457
C03591=1205.471,407.051,-82.293,-175.840,8.422,148.457
C03592=1205.467,407.299,-82.328,-175.840,8.425,148.458
C03593=1205.463,407.546,-82.363,-175.838,8.427,148.458
C03594=1205.459,407.794,-82.398,-175.838,8.430,148.459
C03595=1205.454,408.041,-82.433,-175.838,8.432,148.459
C03596=1205.451,408.289,-82.469,-175.838,8.434,148.460
C03597=1205.447,408.537,-82.504,-175.837,8.436,148.460
C03598=1205.442,408.784,-82.539,-175.837,8.438,148.461
C03599=1205.438,409.032,-82.574,-175.837,8.441,148.461
C03600=1205.435,409.279,-82.609,-175.836,8.443,148.462
C03601=1205.430,409.527,-82.644,-175.836,8.445,148.462
C03602=1205.427,409.774,-82.679,-175.835,8.447,148.463
C03603=1205.422,410.021,-82.714,-175.835,8.449,148.463
C03604=1205.418,410.269,-82.749,-175.835,8.452,148.464
C03605=1205.415,410.517,-82.785,-175.835,8.454,148.464
C03606=1205.410,410.764,-82.819,-175.834,8.456,148.464
C03607=1205.406,411.012,-82.855,-175.834,8.458,148.465
C03608=1205.403,411.259,-82.890,-175.834,8.460,148.466
C03609=1205.398,411.506,-82.925,-175.833,8.463,148.466
C03610=1205.395,411.754,-82.960,-175.833,8.465,148.466
C03611=1205.391,412.002,-82.995,-175.833,8.467,148.467
C03612=1205.386,412.249,-83.030,-175.832,8.469,148.467
C03613=1205.383,412.496,-83.066,-175.832,8.472,148.468
C03614=1205.378,412.744,-83.100,-175.831,8.473,148.468
C03615=1205.374,412.991,-83.136,-175.831,8.476,148.469
C03616=1205.371,413.239,-83.171,-175.831,8.478,148.469
C03617=1205.366,413.486,-83.206,-175.830,8.480,148.470
C03618=1205.363,413.734,-83.241,-175.830,8.482,148.470
C03619=1205.359,413.981,-83.277,-175.830,8.485,148.471
C03620=1205.354,414.229,-83.311,-175.830,8.487,148.471
C03621=1205.351,414.476,-83.347,-175.829,8.489,148.472
C03622=1205.347,414.724,-83.383,-175.829,8.491,148.472
C03623=1205.342,414.971,-83.417,-175.829,8.493,148.473
C03624=1205.339,415.219,-83.453,-175.828,8.495,148.473
C03625=1205.335,415.466,-83.488,-175.828,8.498,148.474
C03626=1205.330,415.713,-83.523,-175.828,8.499,148.474
C03627=1205.326,415.961,-83.559,-175.827,8.501,148.474
C03628=1205.321,416.245,-83.599,-175.827,8.504,148.475
C03629=1205.318,416.529,-83.639,-175.826,8.506,148.476
C03630=1205.317,416.813,-83.680,-175.826,8.509,148.476
C03631=1205.318,417.097,-83.719,-175.826,8.511,148.477
C03632=1204.897,417.097,-83.757,-175.829,8.521,148.480
C03633=1204.895,416.810,-83.717,-175.829,8.519,148.480
C03634=1204.897,416.524,-83.676,-175.830,8.517,148.479
C03635=1204.900,416.237,-83.635,-175.830,8.515,148.479
C03636=1204.905,415.950,-83.594,-175.831,8.512,148.478
C03637=1204.909,415.703,-83.559,-175.831,8.510,148.478
C03638=1204.913,415.456,-83.524,-175.831,8.508,148.477
C03639=1204.917,415.208,-83.489,-175.831,8.506,148.477
C03640=1204.921,414.960,-83.453,-175.832,8.504,148.476
C03641=1204.925,414.713,-83.418,-175.832,8.502,148.476
C03642=1204.929,414.465,-83.383,-175.832,8.499,148.475
C03643=1204.933,414.218,-83.348,-175.832,8.497,148.475
C03644=1204.937,413.971,-83.313,-175.833,8.495,148.475
C03645=1204.941,413.723,-83.278,-175.833,8.493,148.474
C03646=1204.944,413.475,-83.242,-175.834,8.491,148.473
C03647=1204.949,413.229,-83.207,-175.834,8.488,148.473
C03648=1204.953,412.981,-83.172,-175.834,8.486,148.473
C03649=1204.956,412.733,-83.137,-175.835,8.484,148.472
C03650=1204.961,412.486,-83.101,-175.835,8.482,148.472
C03651=1204.965,412.238,-83.066,-175.836,8.480,148.471
C03652=1204.969,411.990,-83.031,-175.836,8.478,148.471
C03653=1204.973,411.743,-82.995,-175.836,8.475,148.470
